(* IEC 61131-3 sources: F100R_S278_Temperville/MyController.device.xml.v3^/Plc Logic.plclogic.xml.v3^/Application.application.xml.v3^/02_Operação, 42 files *)

(* ---- A_EncoderCpu.prg.st ---- *)
PROGRAM A_EncoderCpu

// Encoder Mesa do Forno
IF NOT xRunEncoMForno OR xHomeEncoderForno THEN
	xPresetEncoMForno:=TRUE;
ELSE
	xPresetEncoMforno:=FALSE;
END_IF
dValorEncoderForno:=(-1)*dValorEncoderFornoEntrada;

// Encoder Mesa do Resfriamento
IF NOT xRunEncoMResfr OR xHomeEncoderResfriador THEN
	xPresetEncoMResfr:=TRUE;
ELSE
	xPresetEncoMResfr:=FALSE;
END_IF
dValorEncoderResfriador:=(1)*dValorEncoderResfrEntrada;

// Encoder Dutos Resfriador Superior
IF NOT xRunEncoResfrSup02 OR xHomeEncoderDuctosResfriadorSup02 THEN
	xPresetEncoResfrSup02:=TRUE;
ELSE
	xPresetEncoResfrSup02:=FALSE;
END_IF
dValorEncoderDuctosResfriadorSup02:=(1)*dValorEncoderDuctosResfrSup02Entrada;

// Encoder Dutos Resfriador Inferior
(*IF NOT xRunEncoResfrInf02 OR xHomeEncoderDuctosResfriadorInf02 THEN
	xPresetEncoResfrInf02:=TRUE;
ELSE
	xPresetEncoResfrInf02:=FALSE;
END_IF
dValorEncoderDuctosResfriadorInf02:=(-1)*dValorEncoderDuctosResfrInf02Entrada;
*)
// Encoder Dutos Passagem Superior
(*IF NOT xRunEncoResfrSup01 OR xHomeEncoderDuctosResfriadorSup01 THEN
	xPresetEncoResfrSup01:=TRUE;
ELSE
	xPresetEncoResfrSup01:=FALSE;
END_IF
dValorEncoderDuctosResfriadorSup01:=(1)*dValorEncoderDuctosResfrSup01Entrada;*)

// Encoder Dutos Passagem Inferior
(*IF NOT xRunEncoResfrInf01 OR xHomeEncoderDuctosResfriadorInf01 THEN
	xPresetEncoResfrInf01:=TRUE;
ELSE
	xPresetEncoResfrInf01:=FALSE;
END_IF
dValorEncoderDuctosResfriadorInf01:=(1)*dValorEncoderDuctosResfrInf01Entrada;*)

// Encoder Guilhotina 01
(*IF NOT xRunEncoGuilhotina01 OR xHomeEncoderGuilhotinaResfriador01 THEN
	xPresetEncoGuilhotina01:=TRUE;
ELSE
	xPresetEncoGuilhotina01:=FALSE;
END_IF
dValorEncoderGuilhotinaResfriador01:= (-1)*dValorEncoderGuilhoResfr01Entrada;
*)
// Encoder Guilhotina 01 Superior - Passagem
(*IF NOT xRunEncoGuilhotina01Sup OR xHomeEncoderGuilhotinaResfriador01Sup THEN
	xPresetEncoGuilhotina01Sup:=TRUE;
ELSE
	xPresetEncoGuilhotina01Sup:=FALSE;
END_IF
dValorEncoderGuilhotinaResfriador01Sup:= (1)*dValorEncoderGuilhoResfr01SupEntrada;*)

// Encoder Guilhotina 01 Inferior - Passagem
(*IF NOT xRunEncoGuilhotina01Inf OR xHomeEncoderGuilhotinaResfriador01Inf THEN
	xPresetEncoGuilhotina01Inf:=TRUE;
ELSE
	xPresetEncoGuilhotina01Inf:=FALSE;
END_IF
dValorEncoderGuilhotinaResfriador01Inf:= (1)*dValorEncoderGuilhoResfr01InfEntrada;*)

// Encoder Guilhotina 02
IF NOT xRunEncoGuilhotina02 OR xHomeEncoderGuilhotinaResfriador02 THEN
	xPresetEncoGuilhotina02:=TRUE;
ELSE
	xPresetEncoGuilhotina02:=FALSE;
END_IF
dValorEncoderGuilhotinaResfriador02:= (-1)*dValorEncoderGuilhoResfr02Entrada;

(* ---- A_PrincipalOperacao.prg.st ---- *)
PROGRAM A_PrincipalOperacao
VAR
	HabDesabMotorDuctosInf01: HabilitaDesabilita;
	HabDesabMotorDuctosSup01: HabilitaDesabilita;
	HabDesabMotorDuctosInf02: HabilitaDesabilita;
	HabDesabMotorDuctosSup02: HabilitaDesabilita;
	HabDesabMotorGuilho01: HabilitaDesabilita;
	HabDesabMotorGuilho02: HabilitaDesabilita;

	HabDesabMotorGuilho01Sup: HabilitaDesabilita;
	HabDesabMotorGuilho01Inf: HabilitaDesabilita;
END_VAR

//EncoderMForno();
//EncoderMResfr();
//EncoderResfriInf01();
//EncoderResfriSup01();
//EncoderResfriInf02();
//EncoderResfriSup02();
EncoderModulo01();
EncoderModulo02();
//EncoderModulo03();
//EncoderModulo04();
A_EncoderCpu();
B_Receita();
B_Velocidades();
C_ComandosOperacao();
D_SensoresEntrada();
E_MesaEntrada();
F_BufferForno();
F_MesaForno();
G_BufferResfriamento();
G_BufferTemperaPass();
H_MesaPassagem();
H_MesaResfriador();
H1_Dutos_Oscilantes();
I_MesaSaida();
//J_DuctosResfriadorInf01();
//J_DuctosResfriadorSup01();
//J_DuctosResfriadorInf02();
//J_DuctosResfriadorSup02();
//K_Guilhotina01();
//K_Guilhotina01Sup();
//K_Guilhotina01Inf();
//K_Guilhotina02();
L_EstagiosResfriador();
M_Ventilador01();
//M_Ventilador02();
M_Ventilador03();
//M_Ventilador04();
N_Grades();
//N_MesaBasculante();
O_Portas();
P_ComandosEventos();
//Q_Conveccao();
R_Pressostato();
R_PressostatoAnal();
R_ManometroDifusor();
R_SensorVibracao();
S_ElevacaoForno();
//T_Damper();
T_VenezianaDutPass();
T_VenezianaVentInfPass();
V_VentilacaoPainel();
//X_LimpaResfriador02();

//Habilita/Desabilita Resfriador Inferior 01
(*HabDesabMotorDuctosInf01(Entrada:= xBtDuctosInf01Enable,StatusSaida=> xDuctosInf01Enable);
IF xBtDuctosInf01Enable THEN
	xBtDuctosInf01Enable:=FALSE;
END_IF

IF NOT xDuctosInf01Enable THEN
	J_DuctosResfriadorInf01();
END_IF

xDuctosInf01CheckOk:= xDuctosInf01Enable OR xHomeDuctosResfriadorInf01Ok;
*)

// Habilita/Desabilita Resfriador Superior 01
(*HabDesabMotorDuctosSup01(Entrada:= xBtDuctosSup01Enable,StatusSaida=> xDuctosSup01Enable);
IF xBtDuctosSup01Enable THEN
	xBtDuctosSup01Enable:=FALSE;
END_IF

IF NOT xDuctosSup01Enable THEN
	J_DuctosResfriadorSup01();
END_IF

xDuctosSup01CheckOk:= xDuctosSup01Enable OR xHomeDuctosResfriadorSup01Ok;
*)
// Habilita/Desabilita Resfirador Inferior 02
(*HabDesabMotorDuctosInf02(Entrada:= xBtDuctosInf02Enable,StatusSaida=> xDuctosInf02Enable);
IF xBtDuctosInf02Enable THEN
	xBtDuctosInf02Enable:=FALSE;
END_IF

IF NOT xDuctosInf02Enable THEN
	J_DuctosResfriadorInf02();
END_IF

xDuctosInf02CheckOk:= xDuctosInf02Enable OR xHomeDuctosResfriadorInf02Ok;
*)

// Habilita/Desabilita Resfriador Superior 02
HabDesabMotorDuctosSup02(Entrada:= xBtDuctosSup02Enable,StatusSaida=> xDuctosSup02Enable);
IF xBtDuctosSup02Enable THEN
	xBtDuctosSup02Enable:=FALSE;
END_IF

IF NOT xDuctosSup02Enable THEN
	J_DuctosResfriadorSup02();
END_IF

xDuctosSup02CheckOk:= xDuctosSup02Enable OR xHomeDuctosResfriadorSup02Ok;

// Habilita/Desabilita Guilhotina Resfriador 01
(*HabDesabMotorGuilho01(Entrada:= xBtGuilhotina01Enable,StatusSaida=> xGuilhotina01Enable);
IF xBtGuilhotina01Enable THEN
	xBtGuilhotina01Enable:=FALSE;
END_IF

IF NOT xGuilhotina01Enable THEN
	K_Guilhotina01();
END_IF

xGuilhotina01CheckOk:= xGuilhotina01Enable OR xHomeGuilhotina01Ok;
*)
// Habilita/Desabilita Guilhotina Resfirador 02
HabDesabMotorGuilho02(Entrada:= xBtGuilhotina02Enable,StatusSaida=> xGuilhotina02Enable);
IF xBtGuilhotina02Enable THEN
	xBtGuilhotina02Enable:=FALSE;
END_IF

IF NOT xGuilhotina02Enable THEN
	K_Guilhotina02();
END_IF

xGuilhotina02CheckOk:= xGuilhotina02Enable OR xHomeGuilhotina02Ok;

// Habilita/Desabilita Guilhotina Superior Resfirador 01
(*HabDesabMotorGuilho01Sup(Entrada:= xBtGuilhotina01SupEnable,StatusSaida=> xGuilhotina01SupEnable);
IF xBtGuilhotina01SupEnable THEN
	xBtGuilhotina01SupEnable:=FALSE;
END_IF

IF NOT xGuilhotina01SupEnable THEN
	K_Guilhotina01Sup();
END_IF

xGuilhotina01SupCheckOk:= xGuilhotina01SupEnable OR xHomeGuilhotina01SupOk;*)

// Habilita/Desabilita Guilhotina Inferior Resfirador 01
(*HabDesabMotorGuilho01Inf(Entrada:= xBtGuilhotina01InfEnable,StatusSaida=> xGuilhotina01InfEnable);
IF xBtGuilhotina01InfEnable THEN
	xBtGuilhotina01InfEnable:=FALSE;
END_IF

IF NOT xGuilhotina01InfEnable THEN
	K_Guilhotina01Inf();
END_IF

xGuilhotina01InfCheckOk:= xGuilhotina01InfEnable OR xHomeGuilhotina01InfOk;*)

(* ---- B_Receita.prg.st ---- *)
PROGRAM B_Receita
VAR
	TempoEnvioReceita: TON;
	TempoEnvioReceitaIn: BOOL;
	TempoEnvioReceitaQ: BOOL;
	Index: UINT;
	IndexSoma1: UINT;
	IndexSoma2: UINT;
	IndexSoma3: UINT;
	iSomaRecTemperaturaInferior: INT;
	iSomaRecTemperaturaSuperior: INT;
	iSomaRecPorcentagemInferior: INT;
	iSomaRecPorcentagemSuperior: INT;
	iSomaRecVelocidade01Ventilador01: INT;
	iSomaRecVelocidade02Ventilador01: INT;
	iSomaRecVelocidade01Ventilador02: INT;
	iSomaRecVelocidade02Ventilador02: INT;
	iSomaRecVelocidade01Ventilador03: INT;
	iSomaRecVelocidade02Ventilador03: INT;
	iSomaRecVelocidade01Ventilador04: INT;
	iSomaRecVelocidade02Ventilador04: INT;
	dSomaReceitaSuper: DINT;
END_VAR

IF iHabilitaEscritaReceita=1 THEN
	xReceitaCarregadaOk:=FALSE;
	iEscreverReceita:=1;
	TempoEnvioReceitaIn:=TRUE;
	xBloqueioCargaEnvioRec:=TRUE;
	iHabilitaEscritaReceita:=0;

END_IF

IF iEscreverReceita=1 THEN
	IF 	sEntradaNomedaReceita=sRecNomedaReceita THEN
			xEntradaReenvioRec:=TRUE;
	ELSE
			xEntradaReenvioRec:=FALSE;
	END_IF

	iEntradaEspessuraVidro:=iRecEspessuraVidro;
	rBufferEmissividade:=rRecEmissividade;
	// Parametros de Aquecimento

	rBufferSetTemperaturaInferiorGeral:=rRecTemperaturaInferiorGeral;
	rBufferSetTemperaturaSuperiorGeral:=rRecTemperaturaSuperiorGeral;
	rBufferSetPorcentagemInferiorGeral:=rRecPorcentagemInferiorGeral;
	rBufferSetPorcentagemSuperiorGeral:=rRecPorcentagemSuperiorGeral;

	FOR Index:=1 TO iNumResistencias DO
		rBufferSetTemperaturaSuperior[Index]:=rRecTemperaturaSuperior[Index];
		rBufferSetTemperaturaInferior[Index]:=rRecTemperaturaInferior[Index];
		rBufferSetPorcentagemSuperior[Index]:=rRecPorcentagemSuperior[Index];
		rBufferSetPorcentagemInferior[Index]:=rRecPorcentagemInferior[Index];
	END_FOR

	iBufferTempoPausaResistInf:=iRecTempoPausaResistInf;
	iBufferTempoPausaResistSup:=iRecTempoPausaResistSup;
	iBufferTempoPausa02ResistSup:=iRecTempoPausa02ResistSup;
	iBufferTempoInicioPausa02ResistSup:=iRecTempoInicioPausa02ResistSup;

	iBufferTempoConveccao:=iRecTempoConveccao;

	// Parametros da Mesa do Forno
	iBufferTempoDelayCarga:=iRecTempoDelayCarga;
	iBufferTempoPausaRoletes:=iRecTempoPausaRoletes;
	iBufferTempoAquecimForno:=iRecTempoAquecimForno;
	iBufferTempoPosicaoForno:=iRecTempoPosicaoForno;//////////
	iBufferTempoVelocidadeForno:=iRecTempoVelocidadeForno;////
	iBufferVelocidade01Vaivem:=iRecVelocidade01Vaivem;////////
	iBufferVelocidade02Vaivem:=iRecVelocidade02Vaivem;////////
	iBufferVelocidade03Vaivem:=iRecVelocidade03Vaivem;////////
	iBufferVelocidadeCargaMesadoForno:=iRecVelocidadeCargaMesaForno;////////
	iBufferVelocidadeDescargaMesadoForno:=iRecVelocidadeDescargaMesaForno;/////////
	iBufferCorretorCargaMesaEntrada:=iRecCorretorCargaMesaEntrada;////////

	// Parametros da Mesa do Resfriador

	iBufferTempoResfriamento:=iRecTempoResfriamento;
	iBufferTempoTrocaEstagioResfriamento:=iRecTempoTrocaEstagioResfriamento;
	iBufferTempoTrocaEstagio02Resfriamento:=iRecTempoTrocaEstagio02Resfriamento;

	iBufferVelocidade01Ventilador01:=iRecVelocidade01Ventilador01;
	iBufferVelocidade02Ventilador01:=iRecVelocidade02Ventilador01;
	iBufferVelocidade03Ventilador01:=iRecVelocidade03Ventilador01;

	iBufferVelocidade01Ventilador02:=iRecVelocidade01Ventilador02;
	iBufferVelocidade02Ventilador02:=iRecVelocidade02Ventilador02;
	iBufferVelocidade03Ventilador02:=iRecVelocidade03Ventilador02;

	iBufferVelocidade01Ventilador03:=iRecVelocidade01Ventilador03;
	iBufferVelocidade02Ventilador03:=iRecVelocidade02Ventilador03;
	iBufferVelocidade03Ventilador03:=iRecVelocidade03Ventilador03;

	iBufferVelocidade01Ventilador04:=iRecVelocidade01Ventilador04;
	iBufferVelocidade02Ventilador04:=iRecVelocidade02Ventilador04;
	iBufferVelocidade03Ventilador04:=iRecVelocidade03Ventilador04;

	// Parametros Resfriador 01 Inferior
	iBufferValAltura01ResfriadorInf01:=iRecAltura01ResfriadorInf01;
	iBufferValAltura02ResfriadorInf01:=iRecAltura02ResfriadorInf01;
	iBufferValAltura03ResfriadorInf01:=iRecAltura03ResfriadorInf01;

	// Parametros Resfriador 01 Superior
	iBufferValAltura01ResfriadorSup01:=iRecAltura01ResfriadorSup01;
	iBufferValAltura02ResfriadorSup01:=iRecAltura02ResfriadorSup01;
	iBufferValAltura03ResfriadorSup01:=iRecAltura03ResfriadorSup01;
	iBufferVeneziana:=iRecVeneziana;
	iBufferPassagem:=iRecPassagem;

	// Parametros Resfriador 02 Inferior
	iBufferValAltura01ResfriadorInf02:=iRecAltura01ResfriadorInf02;
	iBufferValAltura02ResfriadorInf02:=iRecAltura02ResfriadorInf02;
	iBufferValAltura03ResfriadorInf02:=iRecAltura03ResfriadorInf02;

	// Parametros Resfriador 02 Superior
	iBufferValAltura01ResfriadorSup02:=iRecAltura01ResfriadorSup02;
	iBufferValAltura02ResfriadorSup02:=iRecAltura02ResfriadorSup02;
	iBufferValAltura03ResfriadorSup02:=iRecAltura03ResfriadorSup02;

	// Parametros Guilhotina 01
	iBufferAlturaGhilhotina01:=iRecAlturaGhilhotina01;

	iBufferAlturaGhilhotina01Sup:=iRecAlturaGhilhotina01Sup;
	iBufferAlturaGhilhotina01Inf:=iRecAlturaGhilhotina01Inf;

	// Parametros Guilhotina 02
	iBufferAlturaGhilhotina02:=iRecAlturaGhilhotina02;

	iBufferCorretorCargaMesaResfriador:=iRecCorretorCargaMesaResfriador;//////////////
	iBufferVelocidadeVaiVemResfriador:=iRecVelocidadeVaiVemResfriador;////////////////////
	iBufferVelocidadeDescargaMesadoResfriador:=iRecVelocidadeDescargaMesaResfriador;////////
	iBufferCorretorCargaMesaSaida:=iRecCorretorCargaMesaSaida;////////////////////

	iRecAjustaAlturaDuctosInf01:=iRecAjustaAlturaDuctosInf01;
	iRecAjustaAlturaDuctosSup01:=iRecAjustaAlturaDuctosSup01;
	iRecAjustaAlturaDuctosInf02:=iRecAjustaAlturaDuctosInf02;
	iRecAjustaAlturaDuctosSup02:=iRecAjustaAlturaDuctosSup02;
	iRecAjustaAlturaGuilho01:=iRecAjustaAlturaGuilho01;
	iRecAjustaAlturaGuilho02:=iRecAjustaAlturaGuilho02;

// Conferencia da Receita
	iSomaRecTemperaturaInferior:=0;
	FOR IndexSoma1:=1	TO iNumResistencias DO
		iSomaRecTemperaturaInferior:=iSomaRecTemperaturaInferior + REAL_TO_INT (rRecTemperaturaInferior[IndexSoma1]);
	END_FOR
	iSomaRecPorcentagemInferior:=0;
	FOR IndexSoma2:=1	TO iNumResistencias DO
		iSomaRecPorcentagemInferior:=iSomaRecPorcentagemInferior + REAL_TO_INT (rRecPorcentagemInferior[IndexSoma2]);
	END_FOR
	iSomaRecTemperaturaSuperior:=0;
	iSomaRecPorcentagemSuperior:=0;
	FOR IndexSoma3:=1	TO iNumResistencias DO
		iSomaRecTemperaturaSuperior:=iSomaRecTemperaturaSuperior + REAL_TO_INT (rRecTemperaturaSuperior[IndexSoma3]);
		iSomaRecPorcentagemSuperior:=iSomaRecPorcentagemSuperior + REAL_TO_INT (rRecPorcentagemSuperior[IndexSoma3]);
	END_FOR

iSomaRecVelocidade01Ventilador01:=iRecVelocidade01Ventilador01/10;
iSomaRecVelocidade02Ventilador01:=iRecVelocidade02Ventilador01/10;
iSomaRecVelocidade01Ventilador02:=iRecVelocidade01Ventilador02/10;
iSomaRecVelocidade02Ventilador02:=iRecVelocidade02Ventilador02/10;
iSomaRecVelocidade01Ventilador03:=iRecVelocidade01Ventilador03/10;
iSomaRecVelocidade02Ventilador03:=iRecVelocidade02Ventilador03/10;
iSomaRecVelocidade01Ventilador04:=iRecVelocidade01Ventilador04/10;
iSomaRecVelocidade02Ventilador04:=iRecVelocidade02Ventilador04/10;

(*
dSomaReceitaClp:=INT_TO_DINT(iRecEspessuraVidro+ REAL_TO_INT (rRecTemperaturaInferiorGeral+rRecTemperaturaSuperiorGeral+
rRecPorcentagemInferiorGeral+rRecPorcentagemSuperiorGeral)+iRecTempoPausaResistInf+iRecTempoPausaResistSup+
iRecTempoConveccao+iRecTempoPausaRoletes+iRecTempoAquecimForno+iRecTempoResfriamento+(iSomaRecVelocidade01Ventilador01)+
(iSomaRecVelocidade02Ventilador01)+(iSomaRecVelocidade01Ventilador02)+(iSomaRecVelocidade02Ventilador02)+
iRecTempoTrocaEstagioResfriamento+iRecAltura01Resfriador+iRecAltura02Resfriador+iRecAlturaGhilhotina+
iSomaRecTemperaturaInferior+iSomaRecTemperaturaSuperior+iSomaRecPorcentagemInferior+iSomaRecPorcentagemSuperior);
*)
	dSomaReceitaSuper:=dSomaReceitaSuperClp;

	sEntradaNomedaReceita:=sRecNomedaReceita;
	xFornoReenvioRec:=xEntradaReenvioRec;
	iReceitaEscritaOk:=1;
	iEscreverReceita:=0;
	xEntradaReenvioRec:=0;
	xReceitaCarregadaOk:=TRUE;
	xBloqueioCargaEnvioRec:=FALSE;
	xReceitaEnviadaEventos:=TRUE;
END_IF
(*
TempoEnvioReceita(IN:=TempoEnvioReceitaIn , PT:=T#15S , Q=>TempoEnvioReceitaQ , ET=> );

IF TempoEnvioReceitaQ THEN
	IF dSomaReceitaClp=dSomaReceitaSuper THEN
		iReceitaEscritaOk:=1;
		iEscreverReceita:=0;
		xReceitaCarregadaOk:=TRUE;
		TempoEnvioReceitaIn:=FALSE;
	ELSE
		iReceitaEscritaFalha:=1;
		iEscreverReceita:=0;
		xReceitaCarregadaOk:=FALSE;
		TempoEnvioReceitaIn:=FALSE;
	END_IF
END_IF
*)

IF (iResfriamentoEspessuraVidro=4 OR iResfriamentoEspessuraVidro=5) THEN
	xEspessuraVidroFino:=TRUE;
	xEspessuraVidroGrosso:=FALSE;
	xBufferValvulaDamperDifusor:=TRUE;
ELSE
	xEspessuraVidroFino:=FALSE;
	xEspessuraVidroGrosso:=TRUE;
	xBufferValvulaDamperDifusor:=FALSE;
END_IF

(* ---- B_Velocidades.prg.st ---- *)
PROGRAM B_Velocidades
VAR
	EntradaForno: EquacaoDaReta;
	FornoPassagem: EquacaoDaReta;
	PassagemResfriamento : EquacaoDaReta;
	ResfriamentoSaida: EquacaoDaReta;
	rVelocidadeMesaEntrada: REAL;
	rVelocidadeCargaMesaForno: REAL;
	rVelocidDescargaMesaForno: REAL;
	rVelocidCargaMesaPassagem: REAL;
	rVelocidDescargaMesaPassagem:REAL;
	rVelocidCargaMesaResfriam: REAL;
	rVelocidDescargaMesaResfr: REAL;
	rVelocidadeMesaSaida: REAL;
	iVelocCargaMesaEntrada: INT;
	iVelocCargaMesaPassagem : INT;
	iVelocCargaResfriador: INT;
	iVelocCargaMesaSaida: INT;
END_VAR

rVelocidadeCargaMesaForno:=INT_TO_REAL(iVelocidadeCargaMesadoForno/1);
rVelocidDescargaMesaForno:=INT_TO_REAL(iVelocidadeDescargaMesadoForno/1);
rVelocidDescargaMesaResfr:=INT_TO_REAL(iVelocidadeDescargaMesadoResfriador/1);

iVelocidadeCargaMesaForno:=REAL_TO_INT(iVelocidadeCargaMesadoForno/10);
iVelocidadeDescargaMesaForno:=REAL_TO_INT(iVelocidadeDescargaMesadoForno/10);
iVelocidadeDescargaMesaResfriador:=REAL_TO_INT(iVelocidadeDescargaMesadoResfriador/10);

EntradaForno(
	rValorY:= rVelocidadeCargaMesaForno/100,
	rPy1:= 25, //Velocidade y1 Inversor Forno
	rPy2:= 45, //Velocidade y2 Inversor Forno
	rPx1:= rVelMesaEntrada25/10, //Velocidade x1 Inversor Entrada
	rPx2:= rVelMesaEntrada45/10, //Velocidade x2 Inversor Entrada
	rValorX=> rVelocidadeMesaEntrada);//Velocidade da Mesa de Entrada

iVelocCargaMesaEntrada:=REAL_TO_INT(rVelocidadeMesaEntrada*10);
iVelocidadeCargaMesaEntrada:=iVelocCargaMesaEntrada+iCorretorCargaMesaEntrada;

FornoPassagem(
	rValorY:= rVelocidDescargaMesaForno/100,
	rPy1:= 25,  //Velocidade y1 Inversor Forno
	rPy2:= 45,  //Velocidade y2 Inversor Forno
	rPx1:= rVelMesaPassagem25/10, //Velocidade x1 Inversor Passagem
	rPx2:= rVelMesaPassagem45/10, //Velocidade x2 Inversor Passagem
	rValorX=> rVelocidCargaMesaPassagem);//Velocidade da Mesa do Resfriamento

iVelocCargaMesaPassagem:=REAL_TO_INT(rVelocidCargaMesaPassagem*10);
iVelocidadeCargaMesaPass:=iVelocCargaMesaPassagem+iCorretorCargaMesaPassagem;

PassagemResfriamento(
	rValorY:= rVelocidDescargaMesaForno/100,
	rPy1:= 25,  //Velocidade y1 Inversor passagem
	rPy2:= 45,  //Velocidade y2 Inversor passagem
	rPx1:= rVelMesaResfriamento25/10, //Velocidade x1 Inversor Resfriador
	rPx2:= rVelMesaResfriamento45/10, //Velocidade x2 Inversor Resfriador
	rValorX=> rVelocidCargaMesaResfriam);//Velocidade da Mesa do Resfriamento

iVelocCargaResfriador:=REAL_TO_INT(rVelocidCargaMesaResfriam*10);
iVelocidadeCargaMesaResfriador:=iVelocCargaResfriador+iCorretorCargaMesaResfriador;

ResfriamentoSaida(
	rValorY:= rVelocidDescargaMesaResfr/10,
	rPy1:= rVelMesaResfriamento25, // Velociade y1 Inversor Resfriador
	rPy2:= rVelMesaResfriamento45, // Velociade y2 Inversor Resfriador
	rPx1:= rVelMesaSaida25, // Velociade x1 Inversor Saída
	rPx2:= rVelMesaSaida45, // Velociade x2 Inversor Saída
	rValorX=> rVelocidadeMesaSaida); // Velocidade da Mesa de Saida

iVelocCargaMesaSaida:=REAL_TO_INT(rVelocidadeMesaSaida);
iVelociadeCargaMesadeSaida:=iVelocCargaMesaSaida+iCorretorCargaMesaSaida;

(* ---- C_ComandosOperacao.prg.st ---- *)
PROGRAM C_ComandosOperacao
VAR
	PassoCmdForno: INT;
	PulsoLedFinalizando: TimerGeneration;
	PulsoLedRestart: TimerGeneration;
	PulsoLedEmEspera: TimerGeneration;
	TonxPausaEmergenciaDelay: TOF;
	TpRestart: TP;
	PulsoPoBtReinicia: PulsoPositivo;
	xLedFornoFinalizando: BOOL;
	xBtRestart: BOOL;
	xPoBtReinicia: BOOL;
	PulsoOperManual: TP;
	PulsoOperAutoma: TP;
	TonOperManual: TON;
	TonOperAutoma: TON;
	TofOperManual: TON;
	TofOperAutoma: TON;

	PulsoPoStartCiclo: PulsoPositivo;
	xFornoEmCicloPulso:	BOOL ;

END_VAR

// SEQUENCIA DE CONTROLE DE OPERAÇÃO

// Seleção Operação ou Stand By

//IF xChStandByOperacao THEN
	xOperacaoHabilitada:=TRUE;
//	xOperacaoStandBy:=FALSE;
(*ELSE
	xOperacaoHabilitada:=FALSE;
	xOperacaoStandBy:=TRUE;
END_IF*)

//Seleção do Modo de Operação Manual ou Automatico
IF xChAutomaticoManual THEN
	xOperacaoManual:=TRUE;
	xOperacaoAutoma:=FALSE;
ELSE
	xOperacaoManual:=FALSE;
	xOperacaoAutoma:=TRUE;
END_IF

PulsoOperManual(IN:= xOperacaoManual, PT:=T#1S , Q=> xPulsoOperacaoManual, ET=> );
PulsoOperAutoma(IN:= xOperacaoAutoma, PT:=T#1S , Q=> xPulsoOperacaoAutoma, ET=> );
TonOperManual(IN:= xOperacaoManual, PT:=T#1S , Q=> xTonOperacaoManual, ET=> );
TonOperAutoma(IN:= xOperacaoAutoma, PT:=T#1S , Q=> xTonOperacaoAutoma, ET=> );
TofOperManual(IN:= xOperacaoManual, PT:=T#1S , Q=> xTofOperacaoManual, ET=> );
TofOperAutoma(IN:= xOperacaoAutoma, PT:=T#1S , Q=> xTofOperacaoAutoma, ET=> );

//Botão de Emergência
xEmergencia:=xBtEmergencia;
// Emergencia para o Supervisório
xBtEmergenciaAcionado:= xBtEmergencia;

IF xEmergencia OR xAlarmeMotorForno THEN
	xPause:=TRUE;
	xRestart:=FALSE;
	xPausaEmergencia:=TRUE;
END_IF
IF NOT xEmergencia THEN
	xPause:=FALSE;
END_IF
(* Reinicio sem Botao Reinicia somente no Reset Alarme *)
IF NOT xEmergencia AND bResetAlmGeral THEN
	xRestart:=TRUE;
	xPausaEmergencia:=FALSE;
ELSE
	xRestart:=FALSE;
END_IF

(* Reinicio com Botão Reinicia Apos Reconhecimento do alarme *)
(*PulsoPoBtReinicia(Entrada:=xBtReinicia, SaidaPulsoPo=>xPoBtReinicia );

IF BtRestart OR xPoBtReinicia THEN
	xBtRestart:=TRUE;
	BtRestart:=FALSE;
ELSE
	xBtRestart:=FALSE;
END_IF

TpRestart(IN:=xBtRestart , PT:=T#500MS , Q=>xBtRestart , ET=> );

IF NOT xEmergencia AND xReleSeguranca AND xBtRestart THEN
	xRestart:=TRUE;
	xPausaEmergencia:=FALSE;
ELSE
	xRestart:=FALSE;
END_IF*)

(*--------- LED RESTART ----------*)

(*PulsoLedRestart.ENABLE:=(xLedStart OR xPausaEmergencia) AND NOT xOperacaoManual;

PulsoLedRestart(ENABLE:= , TIMELOW:=T#500MS , TIMEHIGH:=T#500MS , OUT=>xLedRestart );

(* ----- Informação para Botão Restart do Supervisório -----*)

IF NOT xEmergencia AND xReleSeguranca AND xPausaEmergencia THEN
	xbRestart:=TRUE;
ELSE
	xbRestart:=FALSE;
END_IF*)

TonxPausaEmergenciaDelay(IN:=NOT xReleSeguranca(*xPausaEmergencia*), PT:=T#5000MS , Q=>xPausaEmergenciaTof , ET=> );

(*--------------------------------*)

//Sequencia Ciclo Forno
CASE PassoCmdForno OF

		0:	IF xCmdIniciaCiclo THEN
				PassoCmdForno:=10;
			END_IF

		5:	//xCmdIniciaCiclo:=FALSE;
			PassoCmdForno:=7;

		7: IF xEnergiaOk THEN
				PassoCmdForno:=10;
			ELSE
				PassoCmdForno:=0;
			END_IF

		10: IF xTesteNobreakOk OR xNobreakDesabilitado THEN
				PassoCmdForno:=12;
			END_IF

		12:	uStatusInicioCiclo:=1; // Aguardando Ajustar Dutos
			IF xHomeDuctosResfriadorSup02Ok OR xDuctosSup02Enable THEN
				PassoCmdForno:=15;
			//ELSE
				//PassoCmdForno:=0;
			END_IF

		13:	IF xHomeDuctosResfriadorSup01Ok OR xDuctosSup01Enable THEN
				PassoCmdForno:=15;
			//ELSE
				//PassoCmdForno:=0;
			END_IF

		15:	uStatusInicioCiclo:=2; // Aguardando Ajustar Guilhotina
			IF xHomeGuilhotina02Ok OR xGuilhotina02Enable THEN
				PassoCmdForno:=20;
			//ELSE
				//PassoCmdForno:=0;
			END_IF

		16:	IF xHomeGuilhotina01SupOk OR xGuilhotina01SupEnable THEN
				PassoCmdForno:=17;
			//ELSE
				//PassoCmdForno:=0;
			END_IF

		17:	IF xHomeGuilhotina01InfOk OR xGuilhotina01InfEnable THEN
				PassoCmdForno:=20;
			//ELSE
				//PassoCmdForno:=0;
			END_IF

		20:	uStatusInicioCiclo:=3; // Aguardando Carregar Receita
			IF xReceitaCarregadaOk THEN
				PassoCmdForno:=21;
			//ELSE
				//PassoCmdForno:=0;
			END_IF

		21:	uStatusInicioCiclo:=4; // Aguardando Ligar Resistencias
			IF xLigaResistenciaInferior AND xLigaResistenciaSuperior THEN
				PassoCmdForno:=23;
			//ELSE
				//PassoCmdForno:=0;
			END_IF

		(*22:	uStatusInicioCiclo:=5; // Aguardando Ligar Resistencias Superiores
			IF xLigaResistenciaSuperior THEN
				PassoCmdForno:=23;
			//ELSE
				//PassoCmdForno:=0;
			END_IF*)

		23: uStatusInicioCiclo:=6; // Aguardando Finalizar Aquecimento
			IF uStatusAquecimento=2 THEN // Aquecimento finalizado
				PassoCmdForno:=24;
			//ELSE
				//PassoCmdForno:=0;
			END_IF
			IF xCmFinalizaCiclo OR xSemEnergia THEN(*OR xBtHmiFinalizaCiclo OR xBloqueioAtivo*)
				PassoCmdForno:=40;
			END_IF

		24: xCmdIniciaCiclo:=FALSE;
			xSetTempStandyByInicio:=TRUE;
			PassoCmdForno:=30;

		30:	xFornoEmCiclo:=TRUE;
			IF xCmFinalizaCiclo OR xSemEnergia THEN(*OR xBtHmiFinalizaCiclo OR xBloqueioAtivo*)
				PassoCmdForno:=40;
			END_IF
			IF xAbortaCicloForno THEN
				PassoCmdForno:=200;
			END_IF

		40:	xFornoFinalizando:=TRUE;
			xCmFinalizaCiclo:=FALSE;
			//xBtHmiFinalizaCiclo:=FALSE;
			IF xFornoVazio THEN
				PassoCmdForno:=50;
			END_IF
			IF xAbortaCicloForno THEN
				PassoCmdForno:=200;
			END_IF

		50:	xFornoEmCiclo:=FALSE;
			xFornoFinalizando:=FALSE;
			//xReceitaCarregadaOk:=FALSE;
			xDesligaFimVentilador01:=TRUE;
			xDesligaFimVentilador02:=TRUE;
			xDesligaFimVentilador03:=TRUE;
			xDesligaFimVentilador04:=TRUE;
			PassoCmdForno:=0;

		200:xAbortaCicloForno:=FALSE;
			xFornoFinalizando:=FALSE;
			xBtHmiFinalizaCiclo:=FALSE;
			xFornoEmCiclo:=FALSE;
			xFornoFinalizando:=FALSE;

END_CASE

IF (*NOT xBtFinalizaCiclo OR xBtHmiFinalizaCiclo*)xCmFinalizaCiclo  AND xFornoEmEspera THEN
	//xReceitaCarregadaOk:=FALSE;
	dSomaReceitaClp:=0;
	xReceitaAqiecimCarregadaOk:=FALSE;
	xDesligaFimVentilador01:=TRUE;
	xDesligaFimVentilador02:=TRUE;
	xDesligaFimVentilador03:=TRUE;
	xDesligaFimVentilador04:=TRUE;

	//xBtHmiFinalizaCiclo:=FALSE;
END_IF

xFornoEmEspera:= NOT xFornoEmCiclo AND NOT xFornoFinalizando;

PulsoLedEmEspera(ENABLE:= xFornoEmEspera, TIMELOW:=T#1000MS , TIMEHIGH:=T#1000MS , OUT=>xLedMaqEmEspera );

//xLedMaqEmCiclo:=(xFornoEmCiclo AND NOT xFornoFinalizando) OR xLedFornoFinalizando;

//Sequencia Ciclo Máquina

xMaquinaEmCiclo:= xFornoEmCiclo OR xResfriadorEmCiclo;

xMaquinaEmEspera:= NOT xMaquinaEmCiclo;

// Led Indicação Maquina em Ciclo/Stand-By

PulsoLedFinalizando(ENABLE:= xFornoFinalizando, TIMELOW:=T#500MS , TIMEHIGH:=T#500MS , OUT=>xLedFornoFinalizando );

xLedMaqEmCiclo:=(xFornoEmCiclo AND NOT xFornoFinalizando) OR xLedFornoFinalizando OR xLedMaqEmEspera;

// Libera Ajuste da Altura dos Ductos e da Guilhotina

IF iRecAjustaAlturaDuctosInf01=1 AND xFornoEmCiclo AND xReceitaCarregadaOk THEN
	xBtRecAjustaAlturaDuctosInf01:=TRUE;
	iRecAjustaAlturaDuctosInf01:=0;
END_IF

IF iRecAjustaAlturaDuctosSup01=1 AND xFornoEmCiclo AND xReceitaCarregadaOk THEN
	xBtRecAjustaAlturaDuctosSup01:=TRUE;
	iRecAjustaAlturaDuctosSup01:=0;
END_IF

IF iRecAjustaAlturaDuctosInf02=1 AND xFornoEmCiclo AND xReceitaCarregadaOk THEN
	xBtRecAjustaAlturaDuctosInf02:=TRUE;
	iRecAjustaAlturaDuctosInf02:=0;
END_IF

IF iRecAjustaAlturaDuctosSup02=1 AND xFornoEmCiclo AND xReceitaCarregadaOk THEN
	xBtRecAjustaAlturaDuctosSup02:=TRUE;
	iRecAjustaAlturaDuctosSup02:=0;
END_IF

IF iRecAjustaAlturaGuilho01=1 AND xFornoEmCiclo AND xReceitaCarregadaOk THEN
	xBtRecAjustaGuilhotina01:=TRUE;
	iRecAjustaAlturaGuilho01:=0;
END_IF

IF iRecAjustaAlturaGuilho02=1 AND xFornoEmCiclo AND xReceitaCarregadaOk THEN
	xBtRecAjustaGuilhotina02:=TRUE;
	iRecAjustaAlturaGuilho02:=0;
END_IF

// Auto Home Motores Dutos e Guilhotina
PulsoPoStartCiclo(Entrada:= xFornoEmCiclo, SaidaPulsoPo=> xFornoEmCicloPulso);

IF xFornoEmCicloPulso AND NOT xFornoEmCiclocomCarga AND NOT xResfriadorEmCiclo THEN
	xAutoHomeResfInf02	:= TRUE ;
	xAutoHomeResfSup02	:= TRUE ;
	xAutoHomeGuilho01	:= TRUE ;
	xAutoHomeGuilho02	:= TRUE ;
END_IF

IF xOperacaoManual THEN
	PassoCmdForno:=0;
	xAbortaCicloForno:=FALSE;
	xFornoFinalizando:=FALSE;
	xBtHmiFinalizaCiclo:=FALSE;
	xFornoEmCiclo:=FALSE;
	xFornoFinalizando:=FALSE;
	//xReceitaCarregadaOk:=FALSE;
	dSomaReceitaClp:=0;
	iRecAjustaAlturaDuctosInf01:=0;
	iRecAjustaAlturaDuctosSup01:=0;
	iRecAjustaAlturaDuctosInf02:=0;
	iRecAjustaAlturaDuctosSup02:=0;
	iRecAjustaAlturaGuilho01:=0;
	iRecAjustaAlturaGuilho02:=0;
	xBtRecAjustaAlturaDuctosSup01:=FALSE;
	xBtRecAjustaAlturaDuctosInf01:=FALSE;
	xBtRecAjustaAlturaDuctosSup02:=FALSE;
	xBtRecAjustaAlturaDuctosInf02:=FALSE;
	xBtRecAjustaGuilhotina01:=FALSE;
	xBtRecAjustaGuilhotina02:=FALSE;

	xPausaEmergencia:=FALSE;
	xAutoHomeResfInf02	:= FALSE ;
	xAutoHomeResfSup02	:= FALSE ;
	xAutoHomeGuilho01	:= FALSE ;
	xAutoHomeGuilho02	:= FALSE ;
END_IF

(* ---- E_MesaEntrada.prg.st ---- *)
PROGRAM E_MesaEntrada
VAR
	PassoMesaEntrada: INT;
	PassoPauseEntrada: INT;
	PassoAlmEntrada: INT;
	PassoManualEntrada: INT;
	///Blocos Nativos
	PulsaLedCarga: TimerGeneration;
	PulsoRetornaSensor: TOF;
	TempoLimRetornoSensor: TON;
	TonDelayMovEntrada: TON;
	TempoDelayCarga: Temporizador;
	TempoAposSairSensor: TON;
	TempoAposSairSensorIn: BOOL;
	TempoAposSairSensorQ: BOOL;
	TonAbortaCargaVazio: TON;
	TonAbortaCargaVazioIn: BOOL;
	TonAbortaCargaVazioQ: BOOL;
	PulsaLedCargaIn: BOOL;
	PulsaLedCargaQ: BOOL;
	///Blocos Criados
	PulsoPoChAvanco: PulsoPositivo;
	PulsoNeChAvanco: PulsoNegativo;
	xChAvancaMesaEntradaPo: BOOL;
	xChAvancaMesaEntradaNe: BOOL;
	xAvancoMesaEntrada: BOOL;
	xRecuoMesaEntrada: BOOL;
	xAvancoJogMesaEntrada: BOOL;
	xRecuoJogMesaEntrada: BOOL;
	xCmdAvancoMesaEntrada: BOOL;
	xCarregaFornoManual: BOOL;
	xCarregaFornoAuto: BOOL;
	///xCarregamentoHabilitado: BOOL;
	xLigaCargaForno: BOOL;
	xCarregandoMesaEntrada: BOOL;
	xSeguraCarga: BOOL;
	xCarregaForno: BOOL;
	xRetornoSensor: BOOL;
	xFornoProntoReceber: BOOL;
	iVelocidadeMesaEntrada: INT;
	///xCargaFornoEmAutomatico: BOOL;
	xCargaFornoEmManual: BOOL;
	xPulsoRetornaSensor: BOOL;
	xDelayMovEntrada: BOOL;
	xFimDelayCarregamento: BOOL;
	xDelayCargaOn: BOOL;
	xTempoDiferencaCargas: BOOL;
	xDesligaCargaVazia: BOOL;
	RPM: INT;
	HZ: INT;
END_VAR

// JOG DA MESA DE ENTRADA
(*Avanço*)
PulsoPoChAvanco(Entrada:= xChAvancaMesaEntrada, SaidaPulsoPo=>xChAvancaMesaEntradaPo );
PulsoNeChAvanco(Entrada:= xChAvancaMesaEntrada, SaidaPulsoNe=>xChAvancaMesaEntradaNe );

xCmdAvancoMesaEntrada:=(xChAvancaMesaEntradaPo OR xCmdAvancoMesaEntrada) AND NOT xChAvancaMesaEntradaNe AND NOT xSensorEntrada;

IF xCmdAvancoMesaEntrada AND NOT xCarregandoForno AND NOT xRetornandoForno AND NOT xSensorEntrada (*AND NOT xPausaEmergencia*) AND xTonOperacaoAutoma THEN
	xAvancoJogMesaEntrada:=TRUE;
ELSE
	xAvancoJogMesaEntrada:=FALSE;
END_IF

PulsoRetornaSensor(IN:=xChAvancaMesaEntradaPo , PT:=T#100MS , Q=>xPulsoRetornaSensor , ET=> );
IF (xPulsoRetornaSensor OR xBtHabilitaCarregamento OR xRecargaForno) AND xSensorEntrada  THEN
	xRetornoSensor:=TRUE;
(*ELSE
	xRetornoSensor:=FALSE;*)
END_IF
// Tempo Limite de retorno pelo sensor
TempoLimRetornoSensor(IN:=xRetornoSensor, PT:=T#6S , Q=> , ET=> );

TempoAposSairSensorIn:=NOT xSensorEntrada;
TempoAposSairSensor(IN:=TempoAposSairSensorIn, PT:=T#3S , Q=>TempoAposSairSensorQ , ET=> );

IF TempoAposSairSensorQ OR TempoLimRetornoSensor.Q  THEN
	xRetornoSensor:=FALSE;
END_IF

(*Recuo*)
IF (xChRecuaMesaEntrada OR xRetornoSensor) AND NOT xCarregandoForno AND NOT xRetornandoForno (*AND NOT xPausaEmergencia*) THEN
	xRecuoJogMesaEntrada:=TRUE;
ELSE
	xRecuoJogMesaEntrada:=FALSE;
END_IF

//PRE CONDIÇÕES PARA CARREGAMENTO
(*xTempoDiferencaCargas*)
// Tempo de Restante de Resfriamento Maior que Programado de Forno -> Segura Carregamento
IF (iTempoResfriamentoRestante>=iTempoAquecimForno-10 ) THEN
	xTempoDiferencaCargas:=TRUE;
ELSE
	xTempoDiferencaCargas:=FALSE;
END_IF
IF xTempoDiferencaCargas AND xResfriadorEmCiclo(*xResfriadorCheio*) THEN
	xSeguraCarga:= TRUE;
ELSE
	xSeguraCarga:= FALSE;
END_IF;
// Habilita Carregamento Automatico
IF xBtHabilitaCarregamento AND xFornoEmCiclo AND NOT xBloqueioCargaEnvioRec AND NOT xFornoFinalizando AND NOT xAvancoJogMesaEntrada AND NOT xRecuoJogMesaEntrada AND NOT xSensorEntrada (**)AND NOT xAlarmeMotorForno (**)AND NOT xAlarmeMotorEntrada THEN
	xCarregamentoHabilitado:=TRUE;
	xCargaFornoEmAutomatico:=TRUE;

END_IF
// Carregamento Manual
IF xBtHabilitaCarregamento AND xFornoEmCiclo AND NOT xBloqueioCargaEnvioRec AND NOT xFornoFinalizando AND xFornoVazio THEN
	xCarregaFornoManual:=TRUE;

END_IF

IF xRecargaForno AND xCarregamentoHabilitado AND NOT xSensorEntrada THEN
	xCarregaFornoAuto:=TRUE;
	xCargaFornoEmAutomatico:=TRUE;
END_IF
IF xRecargaForno THEN
	xRecargaForno:=FALSE;
END_IF

// Tempo de atraso no Carregamento automatico do forno
TempoDelayCarga(
	IniciaTempo:= xDelayCargaForno,
	AbortaTempo:= xOperacaoManual,
	SetPointTempo:= iTempoDelayCarga,
	FimTempo:= xFimDelayCarregamento,
	TempoDecorrido=> iTempoDelayCargaDecorrido,
	TempoRestante=> );

IF xDelayCargaForno THEN
	xDelayCargaOn:=TRUE;
	xDelayCargaForno:=FALSE;
END_IF

IF xFimDelayCarregamento THEN
	xDelayCargaOn:=FALSE;
END_IF

IF (xCarregaFornoAuto OR xCarregaFornoManual) AND NOT  xSeguraCarga AND NOT xDelayCargaOn AND (sEntradaNomedaReceita=sFornoNomedaReceita) THEN
	xCarregaForno:=TRUE;
	xCarregaFornoAuto:=FALSE;
	xCarregaFornoManual:=FALSE;
END_IF

IF  xCarregaForno AND xCarregamentoHabilitado AND NOT xSeguranca THEN
	xLigaCargaForno:=TRUE;
	xCarregaForno:=FALSE;
	xCarregamentoHabilitado:=FALSE;
	xFimDelayCarregamento:=FALSE;
END_IF
IF xSeguranca THEN
	xLigaCargaForno:=FALSE;
	xCarregaForno:=FALSE;
	xCarregamentoHabilitado:=FALSE;
END_IF

IF NOT xCarregandoForno AND xFornoEmCiclo AND NOT xBloqueioCargaEnvioRec AND NOT xFornoFinalizando (**)AND NOT xAlarmeMotorForno (**)and not xAlarmeMotorEntrada THEN
	xFornoProntoReceber:=TRUE;
ELSE
	xFornoProntoReceber:=FALSE;
END_IF

PulsaLedCarga(ENABLE:= xFornoProntoReceber, TIMELOW:=T#500MS , TIMEHIGH:=T#500MS , OUT=>PulsaLedCargaQ );
xLedCargaForno:=(xCargaFornoEmAutomatico OR PulsaLedCargaQ) AND NOT xCarregandoForno;

xCargaEmAutomatico:=xCargaFornoEmAutomatico;

//Aborta Carregamento Automático
IF (((xAvancoJogMesaEntrada OR xRecuoJogMesaEntrada ) AND NOT  xCarregandoForno AND NOT xRetornandoForno) OR NOT xFornoEmCiclo (*OR xAlarmePortaEntradaForno OR xAlarmeMotorEntrada OR xAlarmeMotorForno*)) AND xIniciaCargaMesaEntrada THEN
	xFornoEmCicloComCarga:=FALSE;//
END_IF
IF ((xAvancoJogMesaEntrada OR xRecuoJogMesaEntrada ) AND NOT  xCarregandoForno AND NOT xRetornandoForno) OR NOT xFornoEmCiclo (*OR xAlarmePortaEntradaForno OR xAlarmeMotorEntrada OR xAlarmeMotorForno*) THEN
	xCarregaFornoAuto:=FALSE;
	xCarregaFornoManual:=FALSE;
	xCarregamentoHabilitado:=FALSE;
	PassoMesaEntrada:=0;
	xCargaFornoEmAutomatico:=FALSE;
    xPortaEntradaForno:=FALSE;
	xIniciaCargaMesaEntrada:=FALSE; //->TASK/MesaForno
	xCarregandoMesaEntrada:=FALSE;
	xLigaCargaForno:=FALSE;//

	xFimCarregamentoMesaEntrada:=FALSE;(**)
	xFimCargaMesaEntrada:=FALSE;(**)
	xRetornaMesaEntrada:=FALSE;(**)

	xRecuoMesaEntrada:=FALSE; (*teste*)
	xFimRetornoMesaEntrada:=FALSE;(*teste*)
	xAvancoMesaEntrada:=FALSE;(*teste*)

END_IF

// SEQUENCIA DE CARREGAMENTO
TonDelayMovEntrada(IN:= xInvMesaEntradaHabilitado, PT:=T#1S , Q=> xDelayMovEntrada, ET=> );

CASE PassoMesaEntrada OF

		0:	IF xLigaCargaForno THEN
				IF xMotorFornoLigado THEN
					PassoMesaEntrada:=1;
				END_IF
				IF xPause THEN
					PassoPauseEntrada:=0;
					PassoMesaEntrada:=200;
				END_IF
				IF xAlarmeMotorEntrada OR xAlarmeMotorForno OR xAlarmeGeralEncoderMeForno THEN
					PassoMesaEntrada:=200;
				END_IF
			END_IF

		1: 	xLigaCargaForno:=FALSE;
			PassoMesaEntrada:=2;

		2:	xFornoEmCicloComCarga:=TRUE;
			PassoMesaEntrada:=3;

		3:	iVelocidadeMesaForno:= iVelocidadeCargaMesaForno;(*Velocidade Carga Forno*)
			PassoMesaEntrada:=4;

		4:	PassoMesaEntrada:=5;

		5:	PassoMesaEntrada:=6;

		6:	IF iVelocidadeCargaMesaForno= iFrequenciaMotorMesaForno THEN
				PassoMesaEntrada:=10;
			ELSE
				PassoMesaEntrada:=2;
			END_IF

		10:	xPortaEntradaForno:=TRUE;
			PassoMesaEntrada:=20;

		20:	IF xSensorPortaEntrada THEN
				PassoMesaEntrada:=30;
			END_IF
			IF xPause THEN
				PassoPauseEntrada:=0;
				PassoMesaEntrada:=200;
			END_IF
			IF xAlarmeMotorEntrada OR xAlarmeMotorForno OR xAlarmeGeralEncoderMeForno OR xAlarmePortaEntradaForno THEN
				PassoMesaEntrada:=200;
			END_IF

		30:	iVelocidadeMesaEntrada:= iVelocidadeCargaMesaEntrada;(*Velocidade Carga Mesa Entrada*)
			PassoMesaEntrada:=31;

		31:	xAvancoMesaEntrada:=TRUE;
			PassoMesaEntrada:=40;

   		40:	IF xCarregandoForno THEN
				PassoMesaEntrada:=50;
			ELSE
				PassoMesaEntrada:=44;
			END_IF

		44:	xIniciaCargaMesaEntrada:=TRUE; //->TASK/MesaForno
			xCarregandoMesaEntrada:=TRUE;
			TonAbortaCargaVazioIn:=TRUE;
			PassoMesaEntrada:=45;

		45:	IF xIniciaCargaForno THEN
				PassoMesaEntrada:=46;
			END_IF
			IF xPause THEN
				PassoPauseEntrada:=0;
				PassoMesaEntrada:=200;
			END_IF
			IF xAlarmeMotorEntrada OR xAlarmeMotorForno OR xAlarmeGeralEncoderMeForno OR xAlarmePortaEntradaForno THEN
				PassoMesaEntrada:=200;
			END_IF
			IF TonAbortaCargaVazioQ  THEN
				PassoMesaEntrada:=200;
			END_IF

		46: TonAbortaCargaVazioIn:=FALSE;
			PassoMesaEntrada:=50;

		50:	IF xFimCarregamentoMesaEntrada THEN //<- TASK/MesaForno //
				PassoMesaEntrada:=55;
			END_IF
			IF xPause THEN
				PassoPauseEntrada:=30;
				PassoMesaEntrada:=300;
			END_IF
			IF xAlarmeMotorEntrada OR xAlarmeMotorForno OR xAlarmeGeralEncoderMeForno OR xAlarmePortaEntradaForno THEN
				PassoAlmEntrada:=30;
				PassoMesaEntrada:=400;
			END_IF

		55:	xAvancoMesaEntrada:=FALSE;
			PassoMesaEntrada:=56;

		56:	xCargaFornoEmAutomatico:=FALSE;
			xLigaCargaForno:=FALSE;
			xFimCarregamentoMesaEntrada:=FALSE;
			xCarregandoMesaEntrada:=FALSE;
			PassoMesaEntrada:=60;

		60: PassoMesaEntrada:=70;

		70:	IF xFimCargaMesaEntrada THEN //<- TASK/MesaForno
				PassoMesaEntrada:=120;
			END_IF;
			IF xRetornaMesaEntrada THEN //<- TASK/MesaForno
				PassoMesaEntrada:=80;
			END_IF

		80:	xLigaCargaForno:=FALSE;
			xRetornaMesaEntrada:=FALSE;
			iVelocidadeMesaEntrada:= 1*iVelocidadeCargaMesaEntrada;(*iVelRetornoMesaEntrada;Velocidade Retorno Mesa Entrada*)
			PassoMesaEntrada:=81;

		81:	xRecuoMesaEntrada:=TRUE;
			PassoMesaEntrada:=90;

		90:	IF xFimRetornoMesaEntrada THEN //<- TASK/MesaForno
				PassoMesaEntrada:=100;
			END_IF
			IF xPause THEN
				PassoPauseEntrada:=80;
				PassoMesaEntrada:=300;
			END_IF
			IF xAlarmeMotorEntrada OR xAlarmeMotorForno OR xAlarmeGeralEncoderMeForno OR xAlarmePortaEntradaForno THEN
				PassoAlmEntrada:=80;
				PassoMesaEntrada:=400;
			END_IF

		100:PassoMesaEntrada:=101;

		101:xRecuoMesaEntrada:=FALSE;
			PassoMesaEntrada:=110;

		110:xFimRetornoMesaEntrada:=FALSE;
		    xPortaEntradaForno:=FALSE;
			PassoMesaEntrada:=0;

		120:xFimCargaMesaEntrada:=FALSE;
		    xPortaEntradaForno:=FALSE;
			PassoMesaEntrada:=0;

		//Alarmes
		200:xRecuoMesaEntrada:=FALSE;
			xAvancoMesaEntrada:=FALSE;
			PassoMesaEntrada:=201;

		201:PassoMesaEntrada:=202;

		202: xLigaCargaForno:=FALSE;
			 xPortaEntradaForno:=FALSE;
			 xFornoEmCicloComCarga:=FALSE;
			 xCargaFornoEmAutomatico:=FALSE;
			 xIniciaCargaMesaEntrada:=FALSE;
			 xCarregandoMesaEntrada:=FALSE;
			 PassoMesaEntrada:=0;

		// Emergência Pausa/Reinicio
		300:xRecuoMesaEntrada:=FALSE;
			xAvancoMesaEntrada:=FALSE;
			PassoMesaEntrada:=301;

		301:PassoMesaEntrada:=302;

		302:IF xRestart THEN
				PassoMesaEntrada:=303;
			END_IF

		303:PassoMesaEntrada:=PassoPauseEntrada;

		// Alarme Motor Parada/Reinicio
		400:xRecuoMesaEntrada:=FALSE;
			xAvancoMesaEntrada:=FALSE;
			PassoMesaEntrada:=401;

		401:PassoMesaEntrada:=402;

		402:IF xRestart AND iCanOpenInverMesaEntraStateOk THEN
				PassoMesaEntrada:=PassoAlmEntrada;
			END_IF

END_CASE

// MOVIMENTAÇÃO PELO COMANDO ENTRADAS DIGITAIS DO INVERSOR
// Comando e Direção
xMotorMesaEntradaAvanco:= xAvancoMesaEntrada OR xAvancoJogMesaEntrada;
xMotorMesaEntradaRecuo:= xRecuoMesaEntrada OR xRecuoJogMesaEntrada;

InversorMesaEntrada.i_xAvanco:=xMotorMesaEntradaAvanco;
InversorMesaEntrada.i_xRecuo:=xMotorMesaEntradaRecuo;

// Velocidade
IF xAvancoJogMesaEntrada OR xRecuoJogMesaEntrada THEN
	IF xRetornoSensor THEN
		InversorMesaEntrada.i_iFreqRef:=50;
	ELSE
		InversorMesaEntrada.i_iFreqRef:=iVelocidadeJogMesaEntrada;
	END_IF
ELSE
	InversorMesaEntrada.i_iFreqRef:=iVelocidadeMesaEntrada;
END_IF
//--------------------------------------------------------------------------\\

IF xOperacaoManual THEN
	PassoMesaEntrada:=0;
	PassoPauseEntrada:=0;
	PassoAlmEntrada:=0;
	xCarregamentoHabilitado:=FALSE;
	xCargaFornoEmAutomatico:=FALSE;
	xCarregaFornoManual:=FALSE;
	xCarregaFornoAuto:=FALSE;
	xCarregaForno:=FALSE;
	xLigaCargaForno:=FALSE;
	xIniciaCargaMesaEntrada:=FALSE;
	xCarregandoMesaEntrada:=FALSE;
	xFimCarregamentoMesaEntrada:=FALSE;
	xFimCargaMesaEntrada:=FALSE;
	xRetornaMesaEntrada:=FALSE;
	xFimRetornoMesaEntrada:=FALSE;
	xDelayCargaForno:=FALSE;
	xFimDelayCarregamento:=FALSE;
	xDelayCargaOn:=FALSE;
	xBloqueioCargaEnvioRec:=FALSE;

	xAvancoJogMesaEntrada:=FALSE;
	xRecuoJogMesaEntrada:=FALSE;
	xAvancoMesaEntrada:=FALSE;
	xRecuoMesaEntrada:=FALSE;

END_IF

TonAbortaCargaVazio(IN:= TonAbortaCargaVazioIn, PT:=T#20S , Q=>  TonAbortaCargaVazioQ, ET=>);
IF TonAbortaCargaVazioQ OR xOperacaoManual THEN
	TonAbortaCargaVazioIn:=FALSE;
END_IF

(* ---- F_BufferForno.prg.st ---- *)
PROGRAM F_BufferForno
VAR
	Index: INT;
	iEscreverReceitaForno: INT;
END_VAR

IF ((sEntradaNomedaReceita<>sFornoNomedaReceita) OR xFornoReenvioRec) AND xFornoVazio THEN
	iEscreverReceitaForno:=1;
END_IF

IF iEscreverReceitaForno=1 THEN
	iFornoEspessuraVidro:=iEntradaEspessuraVidro;
	// Parametros de Aquecimento

	rSetTemperaturaInferiorGeral:=rBufferSetTemperaturaInferiorGeral;
	rSetTemperaturaSuperiorGeral:=rBufferSetTemperaturaSuperiorGeral;
	rSetPorcentagemInferiorGeral:=rBufferSetPorcentagemInferiorGeral;
	rSetPorcentagemSuperiorGeral:=rBufferSetPorcentagemSuperiorGeral;

	rSetTemperaturaInferiorGeralAux:=rBufferSetTemperaturaInferiorGeral;
	rSetTemperaturaSuperiorGeralAux:=rBufferSetTemperaturaSuperiorGeral;
	rSetPorcentagemInferiorGeralAux:=rBufferSetPorcentagemInferiorGeral;
	rSetPorcentagemSuperiorGeralAux:=rBufferSetPorcentagemSuperiorGeral;

	FOR Index:=1	TO iNumResistencias DO
		rSetTemperaturaSuperior[Index]:=rBufferSetTemperaturaSuperior[Index];
		rSetTemperaturaInferior[Index]:=rBufferSetTemperaturaInferior[Index];
		rSetPorcentagemSuperior[Index]:=rBufferSetPorcentagemSuperior[Index];
		rSetPorcentagemInferior[Index]:=rBufferSetPorcentagemInferior[Index];
	END_FOR

	iTempoPausaResistInf:=iBufferTempoPausaResistInf;
	iTempoPausaResistSup:=iBufferTempoPausaResistSup;
	iTempoPausa02ResistSup:=iBufferTempoPausa02ResistSup;
	iTempoInicioPausa02ResistSup:=iBufferTempoInicioPausa02ResistSup;

	iTempoConveccao:=iBufferTempoConveccao;

	// Parametros da Mesa do Forno
	iTempoDelayCarga:=iBufferTempoDelayCarga;
	iTempoPausaRoletes:=iBufferTempoPausaRoletes;
	iTempoAquecimForno:=iBufferTempoAquecimForno;
	iTempoPosicaoForno:=iBufferTempoPosicaoForno;//////////
	iTempoVelocidadeForno:=iBufferTempoVelocidadeForno;////
	iVelocidade01Vaivem:=iBufferVelocidade01Vaivem;////////
	iVelocidade02Vaivem:=iBufferVelocidade02Vaivem;////////
	iVelocidade03Vaivem:=iBufferVelocidade03Vaivem;////////
	iVelocidadeCargaMesadoForno:=iBufferVelocidadeCargaMesadoForno;////////
	iVelocidadeDescargaMesadoForno:=iBufferVelocidadeDescargaMesadoForno;/////////
	iCorretorCargaMesaEntrada:=iBufferCorretorCargaMesaEntrada;////////

	// Parametros da Mesa do Resfriador
	rBuffer02Emissividade:=rBufferEmissividade;

	iBuffer02TempoResfriamento:=iBufferTempoResfriamento;
	iBuffer02TempoTrocaEstagioResfriamento:=iBufferTempoTrocaEstagioResfriamento;
	iBuffer02TempoTrocaEstagio02Resfriamento:=iBufferTempoTrocaEstagio02Resfriamento;

	//iBuffer02Velocidade01Ventilador01:=iBufferVelocidade01Ventilador01;
	iVelocidade01Ventilador01:=iBufferVelocidade01Ventilador01;
	iBuffer02Velocidade02Ventilador01:=iBufferVelocidade02Ventilador01;
	iBuffer02Velocidade03Ventilador01:=iBufferVelocidade03Ventilador01;

	iBuffer02Velocidade01Ventilador02:=iBufferVelocidade01Ventilador02;
	iBuffer02Velocidade02Ventilador02:=iBufferVelocidade02Ventilador02;
	iBuffer02Velocidade03Ventilador02:=iBufferVelocidade03Ventilador02;

	iBuffer02Velocidade01Ventilador03:=iBufferVelocidade01Ventilador03;
	iBuffer02Velocidade02Ventilador03:=iBufferVelocidade02Ventilador03;
	iBuffer02Velocidade03Ventilador03:=iBufferVelocidade03Ventilador03;

	iBuffer02Velocidade01Ventilador04:=iBufferVelocidade01Ventilador04;
	iBuffer02Velocidade02Ventilador04:=iBufferVelocidade02Ventilador04;
	iBuffer02Velocidade03Ventilador04:=iBufferVelocidade03Ventilador04;

	// Parametros Resfriador 01 Inferior
	iBuffer02ValAltura01ResfriadorInf01:=iBufferValAltura01ResfriadorInf01;
	iBuffer02ValAltura02ResfriadorInf01:=iBufferValAltura02ResfriadorInf01;
	iBuffer02ValAltura03ResfriadorInf01:=iBufferValAltura03ResfriadorInf01;

	// Parametros Resfriador 01 Superior
	iBuffer02ValAltura01ResfriadorSup01:=iBufferValAltura01ResfriadorSup01;
	iBuffer02ValAltura02ResfriadorSup01:=iBufferValAltura02ResfriadorSup01;
	iBuffer02ValAltura03ResfriadorSup01:=iBufferValAltura03ResfriadorSup01;
	iBuffer02Veneziana:=iBufferVeneziana;
	iBuffer02Passagem:=iBufferPassagem;

	// Parametros Resfriador 02 Inferior
	iBuffer02ValAltura01ResfriadorInf02:=iBufferValAltura01ResfriadorInf02;
	iBuffer02ValAltura02ResfriadorInf02:=iBufferValAltura02ResfriadorInf02;
	iBuffer02ValAltura03ResfriadorInf02:=iBufferValAltura03ResfriadorInf02;

	// Parametros Resfriador 02 Superior
	iBuffer02ValAltura01ResfriadorSup02:=iBufferValAltura01ResfriadorSup02;
	iBuffer02ValAltura02ResfriadorSup02:=iBufferValAltura02ResfriadorSup02;
	iBuffer02ValAltura03ResfriadorSup02:=iBufferValAltura03ResfriadorSup02;

	// Parametros Guilhotina 01
	iBuffer02AlturaGhilhotina01:=iBufferAlturaGhilhotina01;

	iBuffer02AlturaGhilhotina01Sup:=iBufferAlturaGhilhotina01Sup;
	iBuffer02AlturaGhilhotina01Inf:=iBufferAlturaGhilhotina01Inf;

	// Parametros Guilhotina 02
	iBuffer02AlturaGhilhotina02:=iBufferAlturaGhilhotina02;

	iBuffer02CorretorCargaMesaResfriador:=iBufferCorretorCargaMesaResfriador;
	iBuffer02VelocidadeVaiVemResfriador:=iBufferVelocidadeVaiVemResfriador;
	iBuffer02VelocidadeDescargaMesadoResfriador:=iBufferVelocidadeDescargaMesadoResfriador;
	iBuffer02CorretorCargaMesaSaida:=iBufferCorretorCargaMesaSaida;

	sFornoNomedaReceita:=sEntradaNomedaReceita;
	xResfriamentoReenvioRec:=xFornoReenvioRec;
	iEscreverReceitaForno:=0;
	xFornoReenvioRec:=0;
END_IF

IF iFornoEspessuraVidro = 4 THEN
	xEspessuraVidroFino:=TRUE;
	xEspessuraVidroGrosso:=FALSE;
ELSE
	xEspessuraVidroFino:=FALSE;
	xEspessuraVidroGrosso:=TRUE;
END_IF

(* ---- F_MesaForno.prg.st ---- *)
PROGRAM F_MesaForno
VAR
	///Passo da Execução da Movimentação do Forno
	PassoMesaForno: INT;
	///Passo da Execução da Movimentação do Forno
	PassoIniciaForno: INT;
	PassoAlmIniForno: INT;
	PassoManualForno: INT;
	PassoEmergenciaForno: INT;
	PassoPauseForno: INT;
	PassoAlmMesaForno: INT;
	PassoPauseIniForno: INT;
	PassoVelVaivem: INT;
	////////
	PassoPosVaivem: INT;
	///////
	SetRampasForno: GIATV.SetDriveRamp_ATV;
	TpSairForno: TP;
	TonParadaSemEner: TON;
	TonDelayMovForno: TON;
	TonParadaSemEnerIn: BOOL;
	TonParadaSemEnerQ: BOOL;
	TonParadaSemEnerEt: TIME;
	TonAutoResetMotorForno: TON;
	TonAutoResetMotorFornoIn: BOOL;
	TonAutoResetMotorFornoQ: BOOL;
	TonIniVelStd: TON;
	TonIniVelStdIn: BOOL;
	TonIniVelStdQ: BOOL;
	///Bloco Conta Tempo de Pausa dos Roletes
	TempoPausaRoletes: Temporizador;
	///Bloco Conta Tempo de Permanecia no Forno
	TempoAquecimForno: Temporizador;
	TempoTrocaVelocidade: Temporizador;
	///////////////////////////////////////////
	TempoTrocaPosicao: Temporizador;
	///////////////////////////////////////////
	TamanhoCarga: ComprimentoCarga;
	///Bloco Calcula Posições de Paradas da Carga
	CalculosMesaForno: CalculosForno;
	///Bloco Converte Milimetro em Pulsos
	ConversorMilimPul: MmConversorPulso;
	///Bloco Converte Pulsos em Milimetros
	ConversorPulMilim: PulsoConversorMm;
	///Bloco Seleciona Pulsos para Vidro Fino ou Grosso
	SelecaoPulsos: BlocoSelecaoEspessura;
	xExecutaSetRampasForno: BOOL;
	dAceleracaoMesaForno: DINT;
	dDesaceleracaoMesaForno: DINT;
	dAccMesaForno: DINT;
	dDecMesaForno: DINT;
	///Contador muda posição de parada do VaiVem
	ContadorMudaPos: INT;
	///Variaveis que Habilitam o Inicio do Ciclo de Aquecimento
	///Variáveis Booleanas Auxiliares
	xFimTempoPausaRoletes: BOOL;
	xFimTempoAquecForno: BOOL;
	xFinalizaVaivemForno: BOOL;
	xFimCalculoCarga: BOOL;
	xTamanhoCargaFora: BOOL;
	xTamanhoCargaOk: BOOL;
	xReativaVaivem: BOOL;
	///Variáveis inteiras Auxiliares
	dValEncoVelMinForno: DINT;
	dValEncoCargaForno: DINT;
	dValEncoAvancoForno: DINT;
	dValEncoRecuoForno: DINT;
	dValEncoDescargaForno: DINT;
	dValEncoReferenciaResfriador: DINT;
	dValEncoSemEnergia: DINT;
	dValLiberaCargaForno: DINT;
	dTamanhoAreaUtilForno: DINT;
	dTamanhoMaximoCarga: DINT;
	dTamanhoCarga: DINT;
	///Distancia Restante para o fim do Carregamento (milimetro)
	iValorVelMinimaForno: INT;
	iValorCargaForno: INT;
	iValorOscilacaoForno: INT;
	iValorDescargaForno: INT;
	iTamanhoAreaUtilForno: INT;
	iValMilimetroVelMinForno: INT;
	iValMilimetroCargaForno: INT;
	iValMilimetroAvancoForno: INT;
	iValMilimetroRecuoForno: INT;
	iValMilimetroDescargaForno: INT;
	iValMilimetroAreaUtilForno: INT;
	iValMilimetroTamMaxCarga: INT;
	iValMilimetroReferenciaResfriador: INT;
	xSensorEntradaPo: BOOL;
	PulsoPoSensorEntrada: PulsoPositivo;
	xliberaDescargaForno: BOOL;
	xDelayMovForno: BOOL;
	xForceSaidadoVidro: BOOL;
	///Variáveis internas auxiliares para mundaça de Velocidade e Posição
	dValorAvancoForno: DINT;
	///////////////
	dValorRecuoForno: DINT;
	////////////////
	xVelocidade01VaivemForno: BOOL;
	//////
	xPosicao01VaivemForno: BOOL;
	/////////
	xFimTempoTrocaVelocidade: BOOL;
	//////
	xFimTempoTrocaPosicao: BOOL;
	//////
	xTemperaturaDesliga: BOOL;
	xDesligaMotorForno: BOOL;
	xTempoMvFornoIn: BOOL;
	xTempoMvFornoQ: BOOL;
	TempoMvForno: ton;
	rConsumoInicialCarga_kW: REAL;
END_VAR

//SELEÇÃO DOS PARAMETROS PELA ESPESSURA DO VIDRO
// Parametros de medidas do Forno
SelecaoPulsos(
	xSelecao:= xEspessuraVidroFino,
	iEntrada0101:= iValorVelMinimaFornoVidroFin,
	iEntrada0102:= iValorVelMinimaFornoVidroGro,
	iEntrada0201:= iValorCargaFornoVidroFin,
	iEntrada0202:= iValorCargaFornoVidroGro,
	iEntrada0301:= iValorOscilacaoFornoVidroFin,
	iEntrada0302:= iValorOscilacaoFornoVidroGro,
	iEntrada0401:= iValorDescargaFornoVidroFin,
	iEntrada0402:= iValorDescargaFornoVidroGro,
	iEntrada0501:= iTamanhoAreaUtilFornoVidroFin,
	iEntrada0502:= iTamanhoAreaUtilFornoVidroGro,
	iEntrada0601:= iTamanhoCargaMaxFornoVidroFin,
	iEntrada0602:= iTamanhoCargaMaxFornoVidroGro,
	iEntrada0701:= iTamanahoFornoContratoVidroFin,
	iEntrada0702:= iTamanahoFornoContratoVidroGro,
	iSaida01=> iValorVelMinimaForno,
	iSaida02=> iValorCargaForno,
	iSaida03=> iValorOscilacaoForno,
	iSaida04=> iValorDescargaForno,
	iSaida05=> iTamanhoAreaUtilForno,
	iSaida06=> iTamanhoCargaMaxForno,
	iSaida07=> iTamanhoCargaContrato);

//Parametros de Rampas do Inversor
//Aceleração
IF 	xEspessuraVidroFino THEN
	dAccMesaForno:=dAccMesaFornoVidroFin;
	dDecMesaForno:=dDecMesaFornoVidroFin;
ELSE
	dAccMesaForno:=dAccMesaFornoVidroGro;
	dDecMesaForno:=dDecMesaFornoVidroGro;
END_IF

IF (dAccMesaForno<>dAceleracaoMesaForno) OR (dDecMesaForno<>dDesaceleracaoMesaForno) THEN
	dAceleracaoMesaForno:=dAccMesaForno;
	dDesaceleracaoMesaForno:=dDecMesaForno;
	xExecutaSetRampasForno:=TRUE;
ELSE
	xExecutaSetRampasForno:=FALSE;
END_IF

// CALCULOS DE POSICIONAMENTO
CalculosMesaForno(
	DistanciaVelMinForno:= 	iValorVelMinimaForno,
	DistanciaCargaForno:= 	iValorCargaForno,
	TamanhoAreaUtil:= 		iTamanhoAreaUtilForno,
	TamanhoCargaMaxima:= 	iTamanhoCargaMaxForno,
	TamanhoCarga:= 			iTamanhoCargaAtualForno,
	SetPointVelMinCarga=> 	iValMilimetroVelMinForno,
	SetPointCargaForno=> 	iValMilimetroCargaForno,
	SetPointDescargaForno=> iValMilimetroDescargaForno,
	SetPointAvancaVaiVemForno=> iValMilimetroAvancoForno,
	SetPointRecuaVaiVemForno=> iValMilimetroRecuoForno,
	TamanhoAreaUtilForno=> 	iValMilimetroAreaUtilForno,
	TamanhoCargaMaxForno=> 	iValMilimetroTamMaxCarga);

// CONVERSÃO MILIMETROS EM PULSOS

iValMilimetroReferenciaResfriador:=iValDistanciaReferenciaResfriador;

ConversorMilimPul(
	dPulso:= 82071,
	dMilimetro:= 6192,
	iEntrMilimetro01:= iValMilimetroVelMinForno,
	iEntrMilimetro02:= iValMilimetroCargaForno,
	iEntrMilimetro03:= iValMilimetroAvancoForno,
	iEntrMilimetro04:= iValMilimetroRecuoForno,
	iEntrMilimetro05:= iValorDescargaForno,//iValMilimetroDescargaForno,
	iEntrMilimetro06:= iValMilimetroAreaUtilForno,
	iEntrMilimetro07:= iValMilimetroTamMaxCarga,
	iEntrMilimetro08:= 40,
	iEntrMilimetro09:= iValMilimetroReferenciaResfriador,
	iEntrMilimetro10:= 400,//distancia da porta de saida para liberar a carga
	dSaidaPulso01=> dValEncoVelMinForno,
	dSaidaPulso02=> dValEncoCargaForno,
	dSaidaPulso03=> dValEncoAvancoForno,
	dSaidaPulso04=> dValEncoRecuoForno,
	dSaidaPulso05=> dValEncoDescargaForno,
	dSaidaPulso06=> dTamanhoAreaUtilForno,
	dSaidaPulso07=> dTamanhoMaximoCarga,
	dSaidaPulso08=>	dValEncoSemEnergia,
	dSaidaPulso09=> dValEncoReferenciaResfriador,
	dSaidaPulso10=> dValLiberaCargaForno);

// CALCULO DO TAMANHO DA CARGA

PulsoPoSensorEntrada(Entrada:= xSensorEntrada, SaidaPulsoPo=>xSensorEntradaPo );

IF	xSensorEntradaPo AND xIniciaCargaMesaEntrada THEN
	xIniciaCargaForno:=TRUE;
	xIniciaCargaMesaEntrada:=FALSE;
END_IF

TamanhoCarga(
	Sensor:= xSensorEntrada,
	Habilita:= xCarregandoForno,
	ValEncoder:= dValorEncoderForno,
	FimMedicao:= xFimCalculoCarga,
	TamanhoCarga=> dTamanhoCarga);

// Desligamento pela Temperatura

IF rMediaLogicaTemperaturaTotal< 0 THEN
	xTemperaturaDesliga:=TRUE;
ELSE
	xTemperaturaDesliga:=FALSE;
END_IF

IF xTemperaturaDesliga AND NOT xResistenciasLigadas THEN
	xDesligaMotorForno:=TRUE;
	xDesligaMotorFornoTempBaixa:=TRUE;
ELSE
	xDesligaMotorForno:=FALSE;
	xDesligaMotorFornoTempBaixa:=FALSE;
END_IF

// MOVIMENTAÇÃO DA MESA DO FORNO
// Atrase para iniciar motor após habilitação
TonDelayMovForno(IN:= xInvMesaFornoHabilitado, PT:=T#1S , Q=> xDelayMovForno, ET=> );
TempoMvForno(IN:= xTempoMvFornoIn, PT:=T#2S , Q=> xTempoMvFornoQ, ET=> );

// Movimentação Stand-By
CASE PassoIniciaForno OF

	0:	(*IF xDelayMovForno THEN
			xLedStart:=TRUE;
		END_IF
		IF xRestart THEN
			PassoIniciaForno:=1;
		END_IF

	1:*)  xLedStart:=FALSE;
		IF NOT xFornoEmCicloComCarga (*AND xDelayMovForno AND NOT xErroEixoMf*) AND NOT xOperacaoManual THEN
			PassoIniciaForno:=2;
			PassoManualForno:=0;
		END_IF

	2:	TonIniVelStdIn:=TRUE;
		IF TonIniVelStdQ THEN
			PassoIniciaForno:=3;
		END_IF

	3:	TonIniVelStdIn:=FALSE;
		PassoIniciaForno:=5;

	5:  iVelocidadeMesaForno:= iVelocidadeStbForno;(*Velocidade Stand-By Forno*)
		PassoIniciaForno:=10;

	10:	xAvancoMesaForno:=TRUE;
		PassoIniciaForno:=15;

	15:	IF iVelocidadeMesaForno<> iVelocidadeStbForno THEN
			PassoIniciaForno:=5;
		END_IF
		IF xFornoEmCicloComCarga THEN
			PassoIniciaForno:=20;
		END_IF
		IF	xDesligaMotorForno THEN
			PassoIniciaForno:=100;
		END_IF
		IF xSemEnergia THEN
			PassoIniciaForno:=50;
		END_IF
		IF xPause THEN
			PassoPauseIniForno:=5;
			PassoIniciaForno:=300;
		END_IF
		IF xAlarmeMotorForno THEN
			PassoAlmIniForno:=5;
			PassoIniciaForno:=400;
		END_IF

	20: IF NOT xFornoEmCicloComCarga THEN
			PassoIniciaForno:=0;
		END_IF

	50: xAvancoMesaForno:=FALSE;
		PassoIniciaForno:=55;

	55: PassoIniciaForno:=60;

	60:	TonParadaSemEnerIn:=TRUE;
		IF TonParadaSemEnerQ THEN
			PassoIniciaForno:=63;
		END_IF
		IF xEnergiaOk THEN
			PassoIniciaForno:=90;
		END_IF

	63:	TonParadaSemEnerIn:=FALSE;
		xHomeEncoderForno:=TRUE;
		PassoIniciaForno:=64;

	64: iVelocidadeMesaForno:= iVelocidadeStbForno;(*Velocidade Stand-By Forno*)
		PassoIniciaForno:=65;

	65:	xHomeEncoderForno:=FALSE;
		PassoIniciaForno:=70;

	70:	xAvancoMesaForno:=TRUE;
		PassoIniciaForno:=75;

	75: IF (dValorEncoderForno>=dValEncoSemEnergia) THEN
			PassoIniciaForno:=50;
		END_IF

	90:	TonParadaSemEnerIn:=FALSE;
		PassoIniciaForno:=0;

	100:xAvancoMesaForno:=FALSE;
		PassoIniciaForno:=105;

	105: PassoIniciaForno:=110;

	110: IF NOT xDesligaMotorForno THEN
		    PassoIniciaForno:=0;
	     END_IF

	// Emergência Pausa/Reinicio
	300:xAvancoMesaForno:=FALSE;
		PassoIniciaForno:=301;

	301:PassoIniciaForno:=302;

	302:IF xRestart THEN
			PassoIniciaForno:=303;
		END_IF

	303:PassoIniciaForno:=PassoPauseIniForno;

		// Alarme Motor Parada/Reinicio

	400:xAvancoMesaForno:=FALSE;
		PassoIniciaForno:=401;

	401:TonAutoResetMotorFornoIn:=TRUE;
		IF TonAutoResetMotorFornoQ THEN
			PassoIniciaForno:=402;
		END_IF

	402: xAutoResetMotorForno:=TRUE;
		PassoIniciaForno:=403;

	403: TonAutoResetMotorFornoIn:=FALSE;
		 PassoIniciaForno:=404;

	404:IF (xRestart OR xAutoResetMotorForno) AND iCanOpenInverMesaFornoStateOk  THEN
			xAutoResetMotorForno:=FALSE;
			PassoIniciaForno:=PassoAlmIniForno;
		END_IF

END_CASE
TonAutoResetMotorForno(IN:=TonAutoResetMotorFornoIn , PT:=T#1000MS , Q=>TonAutoResetMotorFornoQ , ET=> );

TonIniVelStd(IN:=TonIniVelStdIn , PT:=T#100MS , Q=>TonIniVelStdQ , ET=> );
TonParadaSemEner(IN:=TonParadaSemEnerIn , PT:=T#1M , Q=>TonParadaSemEnerQ , ET=>TonParadaSemEnerEt );

iTempoPassoSemEnerg:= DINT_TO_INT((TIME_TO_DINT(T#1M))/1000-(TIME_TO_DINT(TonParadaSemEnerEt))/1000);

// Condição para Descarga do Forno
xliberaDescargaForno:= (xAvancandMesaResfriador AND xFinalizaVaivemForno AND xResfriadorVazio(*AND xDuctosSup01CheckOk AND xGuilhotina01CheckOk AND xVelocidadeVentilador01Ok AND xVelocidadeVentilador02Ok AND xVelocidadeVentilador03Ok*)) OR xForceSaidadoVidro;

// Movimentação em Ciclo
// Sequencia de mudança de Velocidade de VaiVem
CASE PassoVelVaivem OF
	0:	IF xVelocidade01VaivemForno THEN
			PassoVelVaivem:=5;
		END_IF

	5:	xVelocidade01VaivemForno:=FALSE;
		PassoVelVaivem:=10;

	10:	iVelocidadeVaiVemMesaForno := REAL_TO_INT(iVelocidade01Vaivem/10);
		IF xFimTempoTrocaPosicao THEN
			PassoVelVaivem:=15;
		END_IF

	15:	iVelocidadeVaiVemMesaForno:= REAL_TO_INT(iVelocidade02Vaivem/10);
		IF xFimTempoTrocaVelocidade THEN
			PassoVelVaivem:=20;
		END_IF

	20: iVelocidadeVaiVemMesaForno:=REAL_TO_INT(iVelocidade03Vaivem/10);
		//PassoVelVaivem:=20;

	//20:	PassoVelVaivem:=0;
END_CASE

// Sequencia de mudança de Posicao de VaiVem
CASE PassoPosVaivem OF
	0:	IF xPosicao01VaivemForno THEN
			PassoPosVaivem:=5;
		END_IF

	5:	xPosicao01VaivemForno:=FALSE;
		PassoPosVaivem:=10;

	10:	IF NOT xFimTempoTrocaPosicao THEN
			IF ContadorMudaPos=0 THEN
				dValorAvancoForno:= dValEncoCargaForno;
				dValorRecuoForno:= dValEncoCargaForno-773;//Recua 50mm
			END_IF
			IF ContadorMudaPos=1 THEN
				dValorAvancoForno:= dValEncoCargaForno-154;// Avança com -10mm da posição inicial
				dValorRecuoForno:= dValEncoCargaForno-927;//Recua 60mm
			END_IF
			IF ContadorMudaPos=2 THEN
				dValorAvancoForno:= dValEncoCargaForno-309;// Avança com -20mm da posição inicial
				dValorRecuoForno:= dValEncoCargaForno-1081;//Recua 70mm;
			END_IF
			IF ContadorMudaPos=3 THEN
				dValorAvancoForno:= dValEncoCargaForno-463;// Avança com -30mm da posição inicial
				dValorRecuoForno:= dValEncoCargaForno-1235;//Recua 80mm;
			END_IF
		ELSE
			xTempoPausaRoletesOn:=FALSE;
			PassoPosVaivem:=15;
		END_IF

	15:	IF ContadorMudaPos=0 THEN
			dValorAvancoForno:= dValEncoAvancoForno;
			dValorRecuoForno:= dValEncoRecuoForno;
		END_IF
		IF ContadorMudaPos=1 THEN
			dValorAvancoForno:= dValEncoAvancoForno-154;
			dValorRecuoForno:= dValEncoRecuoForno-154;
		END_IF
		IF ContadorMudaPos=2 THEN
			dValorAvancoForno:= dValEncoAvancoForno-309;
			dValorRecuoForno:= dValEncoRecuoForno-309;
		END_IF
		IF ContadorMudaPos=3 THEN
			dValorAvancoForno:= dValEncoAvancoForno-463;
			dValorRecuoForno:= dValEncoRecuoForno-463;
		END_IF
		//PassoPosVaivem:=0;

END_CASE

// Sequencia de Entrada, Oscilação e Saída

CASE PassoMesaForno OF

	0:	IF xIniciaCargaForno AND xFornoEmCiclo THEN
			PassoMesaForno:=1;
		END_IF

	1:	xHomeEncoderForno:=TRUE;
		PassoMesaForno:=2;

	2:	xMesaFornoOn:=TRUE;
		PassoMesaForno:=5;

	5:	xHomeEncoderForno:=FALSE;
		PassoMesaForno:=6;

	6:	iVelocidadeMesaForno:= iVelocidadeCargaMesaForno;(*Velocidade Carga Forno*)
		PassoMesaForno:=7;

	7:	xAvancoMesaForno:=TRUE;
		PassoMesaForno:=10;

	10:	xIniciaCargaForno:=FALSE;
		xIniciaCargaMesaEntrada:=FALSE;
		xExecutaMovMesaForno:=FALSE;
		//xPortaEntradaForno:=TRUE;
		xCarregandoForno:=TRUE;
		xStartCargaForno:=TRUE;
		xFornoCheio:=TRUE;
		PassoMesaForno:=20;

	20: IF (dValorEncoderForno>=dValEncoVelMinForno) THEN
			PassoMesaForno:=30;
		END_IF
		IF xPause THEN
			PassoPauseForno:=5;
			PassoMesaForno:=300;
		END_IF
		IF xAlarmeMotorEntrada OR xAlarmeMotorForno OR xAlarmeGeralEncoderMeForno OR xAlarmePortaEntradaForno THEN
			PassoAlmMesaForno:=5;
			PassoMesaForno:=400;
		END_IF

	30: iVelocidadeMesaForno:= iVelMinCargaForno;(*Velocidade Minima Carga Forno*)
		PassoMesaForno:=40;

	40: IF (dValorEncoderForno>=dValEncoCargaForno) THEN
			PassoMesaForno:=42;
		END_IF
		IF xPause THEN
			PassoPauseForno:=5;
			PassoMesaForno:=300;
		END_IF
		IF xAlarmeMotorForno THEN
			PassoAlmMesaForno:=5;
			PassoMesaForno:=400;
		END_IF

	42: iVelocidadeMesaForno:= 0;
		xAvancoMesaForno:=FALSE;
		PassoMesaForno:=45;

	45: IF (iVelocidade01Vaivem=0) AND (iTempoPosicaoForno<>0)THEN
			xTempoPausaRoletesOn:=TRUE;
		END_IF
		PassoMesaForno:=50;

	50: xExecutaMovMesaForno:=FALSE;
		xCarregandoForno:=FALSE;
		xIniciaCargaForno:=FALSE;
		xFimCarregamentoMesaEntrada:=TRUE; //-> TASK/MesaEntrada
		PassoMesaForno:=55;

	55: IF xFimCalculoCarga THEN
			PassoMesaForno:=60;
		END_IF

	60:	IF (dTamanhoCarga>=dTamanhoAreaUtilForno) OR (dTamanhoCarga>dTamanhoMaximoCarga) OR (dTamanhoCarga<=0) OR  (xSensorEntrada) THEN
			xTamanhoCargaFora:=TRUE;
			xRetornaMesaEntrada:=TRUE; //-> TASK/MesaEntrada
			PassoMesaForno:=70;
		END_IF
		IF (dTamanhoCarga<=dTamanhoMaximoCarga) AND NOT xSensorEntrada THEN
			xTamanhoCargaOk:=TRUE;
			xFimCargaMesaEntrada:=TRUE;//-> TASK/MesaEntrada
			PassoMesaForno:=100;
		END_IF

	70:	xTamanhoCargaFora:=FALSE;
		iVelocidadeMesaForno:= 1*iVelocidadeCargaMesaForno;(*iVelRetornoCargaForno;Velocidade de Retorno Forno*)
		PassoMesaForno:=71;

	71:	xRecuoMesaForno:=TRUE;
		PassoMesaForno:=80;

	80:	xRetornandoForno:=TRUE;
		xExecutaMovMesaForno:=FALSE;
		xTempoPausaRoletesOn:=FALSE;
		IF (dValorEncoderForno<=0) THEN
			PassoMesaForno:=90;
		END_IF
		IF xPause THEN
			PassoPauseForno:=70;
			PassoMesaForno:=300;
		END_IF
		IF xAlarmeMotorEntrada OR xAlarmeMotorForno OR xAlarmeGeralEncoderMeForno OR xAlarmePortaEntradaForno THEN
			PassoAlmMesaForno:=70;
			PassoMesaForno:=400;
		END_IF

	90: xFimRetornoMesaEntrada:=TRUE; //-> TASK/MesaEntrada
		xRecuoMesaForno:=FALSE;		(* DesLiga Recuo Motor Pre Forno *)
		xRetornandoForno:=FALSE;
		xFornoCheio:=FALSE;
		xFornoEmCicloComCarga:=FALSE;
		xPortaEntradaForno:=FALSE;
		xMesaFornoOn:=FALSE;
		PassoIniciaForno:=20;
		PassoMesaForno:=0;

	100: uNumeroCargaRel:=uNumeroCargaRel+1;
		 rConsumoInicialCarga_kW:=rConsumoEnergiaReal_kWh;(*Ativo*)
		 PassoMesaForno:=101;

	101:xIniciaRelatorioProd:=TRUE;
		PassoMesaForno:=102;

	102: xTamanhoCargaOk:=FALSE;
		 xPortaEntradaForno:=FALSE;
		 xFornoCarregado:= TRUE;
		 xFornoComCarga:=TRUE;
		 xIniciaPausaResistencias:= TRUE;
		 xPausaHabilitaTesteEncoder:=TRUE;
		 xLigaConveccaoForno:= TRUE;
		 xVelocidade01VaivemForno:=TRUE;////////
		 xPosicao01VaivemForno:=TRUE;///////////
		 PassoMesaForno:=110;

	110://IF 	xFimTempoPausaRoletes THEN
			PassoMesaForno:=120;
		//END_IF
		IF xPause THEN
			PassoPauseForno:=110;
			PassoMesaForno:=300;
		END_IF
		IF xAlarmeMotorForno THEN
			PassoAlmMesaForno:=110;
			PassoMesaForno:=400;
		END_IF

	120:IF ContadorMudaPos>=4 THEN
			 ContadorMudaPos:=0;
		END_IF
		PassoMesaForno:=121;

	121:xPausaHabilitaTesteEncoder:=FALSE;
		iVelocidadeMesaForno:= 1*iVelocidadeVaiVemMesaForno;(*Velocidade Vai Vem Forno*)
		PassoMesaForno:=122;

	122:xRecuoMesaForno:=TRUE;
		PassoMesaForno:=130;

	130:PassoMesaForno:=135;

	135:IF NOT xliberaDescargaForno OR xAlarmePortaSaidaFornoAberta THEN
			IF (dValorEncoderForno<=dValorRecuoForno) THEN
				PassoMesaForno:=140;
			END_IF
			IF iVelocidadeMesaForno <> 1*iVelocidadeVaiVemMesaForno THEN
				PassoMesaForno:=121;
			END_IF
			IF xPause THEN
				PassoPauseForno:=121;
				PassoMesaForno:=300;
			END_IF
			IF xAlarmeMotorForno OR xAlarmeGeralEncoderMeForno THEN
				PassoAlmMesaForno:=121;
				PassoMesaForno:=400;
			END_IF
		ELSE
			IF	(dValorEncoderForno<=dValEncoCargaForno - dValLiberaCargaForno) THEN
					PassoMesaForno:=156;
			END_IF
			IF iVelocidadeMesaForno <> 1*iVelocidadeVaiVemMesaForno THEN
				PassoMesaForno:=121;
			END_IF
			IF xPause THEN
				PassoPauseForno:=121;
				PassoMesaForno:=300;
			END_IF
			IF xAlarmeMotorForno OR xAlarmeGeralEncoderMeForno THEN
				PassoAlmMesaForno:=121;
				PassoMesaForno:=400;
			END_IF
		END_IF

	140:xRecuoMesaForno:=FALSE;
		PassoMesaForno:=141;

	141:xForceSaidadoVidro:=FALSE;
		PassoMesaForno:=145;

	145:iVelocidadeMesaForno:= iVelocidadeVaiVemMesaForno;(*Velocidade Vai Vem Forno*)
		PassoMesaForno:=146;

	146:xAvancoMesaForno:=TRUE;
		PassoMesaForno:=150;

	150:PassoMesaForno:=151;

	151:IF NOT xliberaDescargaForno OR xAlarmePortaSaidaFornoAberta THEN
			IF (dValorEncoderForno>=dValorAvancoForno) THEN
				PassoMesaForno:=155;
			END_IF
			IF iVelocidadeMesaForno <> 1*iVelocidadeVaiVemMesaForno THEN
				PassoMesaForno:=145;
			END_IF
			IF xPause THEN
				PassoPauseForno:=145;
				PassoMesaForno:=300;
			END_IF
			IF xAlarmeMotorForno OR xAlarmeGeralEncoderMeForno THEN
				PassoAlmMesaForno:=145;
				PassoMesaForno:=400;
			END_IF
		ELSE
			IF	(dValorEncoderForno<=dValEncoCargaForno - dValLiberaCargaForno) THEN
				PassoMesaForno:=157;
			ELSE
				PassoMesaForno:=155;
			END_IF
			IF iVelocidadeMesaForno <> 1*iVelocidadeVaiVemMesaForno THEN
				PassoMesaForno:=145;
			END_IF
			IF xPause THEN
				PassoPauseForno:=145;
				PassoMesaForno:=300;
			END_IF
			IF xAlarmeMotorForno OR xAlarmeGeralEncoderMeForno THEN
				PassoAlmMesaForno:=145;
				PassoMesaForno:=400;
			END_IF
		END_IF

	155: xAvancoMesaForno:=FALSE;
		 ContadorMudaPos:=ContadorMudaPos+1;
		 PassoMesaForno:=120;

	156:xRecuoMesaForno:=FALSE;
		xAvancoMesaForno:=TRUE;
		xForceSaidadoVidro:=FALSE;
		PassoMesaForno:=157;

	157:xForceSaidadoVidro:=FALSE;
		PassoMesaForno:=160;

	160://xForceSaidadoVidro:=FALSE;
		PassoMesaForno:=164;

	164:xAvancoMesaForno:=TRUE;
		PassoMesaForno:=165;

	165:iVelocidadeMesaForno:= iVelocidadeDescargaMesaForno;(*Velocidade Descarga Forno*)
		PassoMesaForno:=166;

	166:PassoMesaForno:=170;

	170:IF xDescarregandoForno THEN
			PassoMesaForno:=180;
		ELSE
			PassoMesaForno:=171;
		END_IF

	171:xAbreVenezVentPass:=TRUE;//-> TASK/T_VenezianaVentInfPass
		xPortaSaidaForno:=TRUE;
		xValvulaScanner:=TRUE;
		xDescarregandoForno:=TRUE;
		//xReajustaAlturaDuctosSup02:=TRUE;
		xFornoCarregado:= FALSE;
		xPulsoTrocaParamResfriador:=TRUE;
		xIniciaPausaResistencias:= FALSE;
		xLigaConveccaoForno:= FALSE;
		PassoMesaForno:=172;

	172:IF (dValorEncoderForno>=dValEncoCargaForno) AND xSensorPortaSaida THEN
			PassoMesaForno:=175;
		END_IF
		IF (dValorEncoderForno>=dValEncoCargaForno) AND NOT xSensorPortaSaida THEN
			PassoMesaForno:=173;
		END_IF
		IF xPause THEN
			xDescarregandoForno:=FALSE;
			xFornoCarregado:= TRUE;
			PassoPauseForno:=121;
			PassoMesaForno:=300;
		END_IF
		(*IF xAlarmeMeFornoParado THEN // Só funciona se resetar Este alarme
			xDescarregandoForno:=FALSE;
			xFornoCarregado:= TRUE;
			PassoMesaForno:=121;
		END_IF*)

	173: xDescarregandoForno:=FALSE;
		 xFornoCarregado:= TRUE;
		 xAvancoMesaForno:=FALSE;
		 PassoMesaForno:=120;

	175: //xValvulaScanner:=TRUE;
		 PassoMesaForno:=176;

	176: xFimTempoPausaRoletes:=FALSE;
		 xFimTempoAquecForno:=FALSE;
		 xFinalizaVaivemForno:=FALSE;
		 xFimTempoTrocaVelocidade:=FALSE;//////
		 xFimTempoTrocaPosicao:=FALSE;//////
		 xFimTempoPausaResistInf:=FALSE;
		 xFimTempoPausaResistSup:=FALSE;
		 xFimTempoPausa02ResistSup:=FALSE;
		 PassoVelVaivem:=0;////////
		 PassoPosVaivem:=0;////////
		 PassoMesaForno:=180;

	180:IF (dValorEncoderForno>=dValEncoReferenciaResfriador) THEN
			xIniciaCargaResfriador:=TRUE;//-> TASK/MesaEntrada
			xIniciaCargaPassagem:=TRUE;//-> TASK/MesaEntrada
			PassoMesaForno:=181;
		END_IF
		IF xPause THEN
			PassoPauseForno:=164;
			PassoMesaForno:=300;
		END_IF
		IF xAlarmeMotorForno OR xAlarmeMotorResfriador OR xAlarmePortaSaidaFornoAberta OR xAlarmeGeralEncoderMeForno OR xAlarmeGeralEncoderMeResfriador THEN
			PassoAlmMesaForno:=164;
			PassoMesaForno:=400;
		END_IF

	181:IF (dValorEncoderForno>=dValEncoDescargaForno) THEN
			PassoMesaForno:=190;
		END_IF
		IF xPause THEN
			PassoPauseForno:=164;
			PassoMesaForno:=300;
		END_IF
		IF xAlarmeMotorForno OR xAlarmeMotorResfriador OR xAlarmePortaSaidaFornoAberta OR xAlarmeGeralEncoderMeResfriador THEN
			PassoAlmMesaForno:=164;
			PassoMesaForno:=400;
		END_IF

	190:xFinalizaRelatorioProd:=TRUE;
		xDescarregandoForno:=FALSE;
		xFornoCheio:=FALSE;
		xFornoComCarga:=FALSE;
		xPortaSaidaForno:=FALSE;
		xValvulaScanner:=FALSE;
		xForceSaidadoVidro:=FALSE;
		xFimDescForIniStdBy:=TRUE;
		xResetPid:=TRUE;
		PassoMesaForno:=191;

	191:IF xCarregamentoHabilitado THEN
			xRecargaForno:=TRUE; //->TASK/MesaEntrada
			xDelayCargaForno:=TRUE; //->TASK/MesaEntrada
			PassoMesaForno:=0;
		ELSE
			xFornoEmCicloComCarga:=FALSE;
			xDelayCargaForno:=TRUE; //->TASK/MesaEntrada
			xMesaFornoOn:=FALSE;
			PassoMesaForno:=0;
		END_IF

	// Emergência Pausa/Reinicio
	300:xAvancoMesaForno:=FALSE;
		xRecuoMesaForno:=FALSE;
		PassoMesaForno:=301;

	301:PassoMesaForno:=302;

	302:IF xRestart THEN
			PassoMesaForno:=303;
		END_IF

	303:PassoMesaForno:=PassoPauseForno;

		// Alarme Motor Parada/Reinicio
	400:xAvancoMesaForno:=FALSE;
		xRecuoMesaForno:=FALSE;
		PassoMesaForno:=401;

	401:PassoMesaForno:=402;

	402:IF (xRestart) AND iCanOpenInverMesaFornoStateOk  THEN
			PassoMesaForno:=PassoAlmMesaForno;
		END_IF

END_CASE

//Consumo de Energia por fornada
rConsumoCargaRel:= rConsumoEnergiaReal_kWh-rConsumoInicialCarga_kW;

TpSairForno(IN:=xBtSairForno , PT:=T#500MS , Q=>xSairForno , ET=> );
IF xBtSairForno THEN
	xBtSairForno:=0;
END_IF

IF xSairForno AND NOT xResfriadorCheio AND xFornoComCarga THEN
	xForceSaidadoVidro:=TRUE;
END_IF

// TEMPORIZADORES
TempoPausaRoletes(
	IniciaTempo:= 	xFornoCarregado,
	AbortaTempo:= 	xSairForno OR xOperacaoManual,
	SetPointTempo:= iTempoPausaRoletes,
	FimTempo:= 		xFimTempoPausaRoletes,
	TempoDecorrido=>iTempoPausaRoleteDecorrido,
	TempoRestante=> iTempoPausaRoleteRestante);

TempoAquecimForno(
	IniciaTempo:= xFornoCarregado,
	AbortaTempo:= xSairForno OR xOperacaoManual,
	SetPointTempo:= iTempoAquecimForno,
	FimTempo:= 		xFimTempoAquecForno,
	TempoDecorrido=>iTempoAquecFornoDecorrido,
	TempoRestante=> iTempoAquecFornoRestante);

xFinalizaVaivemForno:=xFimTempoAquecForno;
xLigaCargaResfriador:=xFimTempoAquecForno;
xLigaCargaPassagem:=xFimTempoAquecForno;
xLigaVent01FimForno:=	xFimTempoAquecForno AND NOT xMotorVentilador01Ligado;
xLigaVent02FimForno:=	xFimTempoAquecForno AND NOT xMotorVentilador02Ligado;
xLigaVent03FimForno:=	xFimTempoAquecForno AND NOT xMotorVentilador03Ligado;
xLigaVent04FimForno:=	xFimTempoAquecForno AND NOT xMotorVentilador04Ligado;

/////////////////////////////////////////////////////
TempoTrocaVelocidade(
	IniciaTempo:= xFimTempoTrocaPosicao,(*xFornoCarregado,*)
	AbortaTempo:= xSairForno OR xOperacaoManual,
	SetPointTempo:= iTempoVelocidadeForno,
	FimTempo:= xFimTempoTrocaVelocidade,
	TempoDecorrido=> iTempoTrocaVelocidadeDecorrido,
	TempoRestante=> );

TempoTrocaPosicao(
	IniciaTempo:= xFornoCarregado,
	AbortaTempo:= xSairForno OR xOperacaoManual,
	SetPointTempo:= iTempoPosicaoForno,
	FimTempo:= xFimTempoTrocaPosicao,
	TempoDecorrido=> iTempoTrocaPosicaoDecorrido,
	TempoRestante=> );

//STATUS
xFornoVazio:=NOT xFornoCheio;

// MOVIMENTAÇÃO PELO COMANDO ENTRADAS DIGITAIS DO INVERSOR
// Comando e Direção
xMotorMesaFornoAvanco:= xAvancoMesaForno;
xMotorMesaFornoRecuo:= xRecuoMesaForno;

InversorMesaForno.i_xAvanco:=xMotorMesaFornoAvanco;
InversorMesaForno.i_xRecuo:=xMotorMesaFornoRecuo;

// Velocidade
InversorMesaForno.i_iFreqRef:=iVelocidadeMesaForno;

//------------------------------------------------------------------------\\

IF	uHoraRealTime=21 AND uMinutoRealTime=0 AND uSegundoRealTime=0 THEN
	uNumeroCargaRel:=0;
END_IF

ConversorPulMilim(
	dPulso:= 82071,
	dMilimetro:= 6192,
	dEntradaPulso01:= dTamanhoCarga,
	iSaidaMilimetro01=> iTamanhoCargaAtualForno );

IF xOperacaoManual THEN
	xLedStart:=FALSE;
	PassoIniciaForno:=0;
	PassoPauseIniForno:=0;
	PassoAlmIniForno:=0;
	PassoMesaForno:=0;
	PassoPauseForno:=0;
	PassoAlmMesaForno:=0;

	PassoVelVaivem:=0;////////
	PassoPosVaivem:=0;///////
	ContadorMudaPos:=0;
	xIniciaCargaForno:=FALSE;
	xHomeEncoderForno:=FALSE;
	xCarregandoForno:=FALSE;
	xFornoCheio:=FALSE;
	xFornoEmCicloComCarga:=FALSE;
	xMesaFornoOn:=FALSE;
	xTamanhoCargaFora:=FALSE;
	xTamanhoCargaOk:=FALSE;
	xRetornandoForno:=FALSE;
	xFornoCarregado:= FALSE;
	xIniciaPausaResistencias:= FALSE;
	xLigaConveccaoForno:= FALSE;
	xFimTempoPausaRoletes:=FALSE;
	xFimTempoAquecForno:=FALSE;
	xFimTempoTrocaVelocidade:=FALSE;//////
	xFimTempoTrocaPosicao:=FALSE;//////
	xFinalizaVaivemForno:=FALSE;
	xFimTempoPausaResistInf:=FALSE;
	xFimTempoPausaResistSup:=FALSE;
	xFimTempoPausa02ResistSup:=FALSE;
	xDescarregandoForno:=FALSE;
	xIniciaRelatorioProd:= FALSE;
	xFinalizaRelatorioProd:= FALSE;
	TonParadaSemEnerIn:=FALSE;
	xTempoPausaRoletesOn:=FALSE;
	xFimCalculoCarga:=FALSE;
	xFornoComCarga:=FALSE;
	xPausaHabilitaTesteEncoder:=FALSE;
	xForceSaidadoVidro:=FALSE;
	xVelocidade01VaivemForno:=FALSE;//////
	xPosicao01VaivemForno:=FALSE;/////////
	xAbreVenezVentPass:=FALSE;
	xValvulaScanner:=FALSE;

	xPortaEntradaForno:=FALSE;
	xPortaSaidaForno:=FALSE;

	xAvancoMesaForno:=FALSE;
	xRecuoMesaForno:=FALSE;
END_IF

xDesabFalhInvMesaForno:= NOT xFornoEmCicloComCarga;

(* ---- G_BufferResfriamento.prg.st ---- *)
PROGRAM G_BufferResfriamento
VAR
	Index: INT;
	iEscreverReceitaResfriamento: INT;
END_VAR

//BUFFER PARAMETROS DO RESFRIAMENTO

(*---------------- SISTEMA NOVO --------------------*)

IF ((sFornoNomedaReceita<>sResfriamentoNomedaReceita) OR xResfriamentoReenvioRec) AND NOT xResfriadorEmCiclo THEN
	iEscreverReceitaResfriamento:=1;
END_IF

IF iEscreverReceitaResfriamento=1 THEN
	xResfriamentoReenvioRec:=0;
	iResfriamentoEspessuraVidro:=iFornoEspessuraVidro;

	// Parametros da Mesa do Resfriador
	rEmissividade:=rBuffer02Emissividade;

	iTempoResfriamento:=iBuffer02TempoResfriamento;
	iTempoTrocaEstagioResfriamento:=iBuffer02TempoTrocaEstagioResfriamento;
	iTempoTrocaEstagio02Resfriamento:=iBuffer02TempoTrocaEstagio02Resfriamento;

	//iVelocidade01Ventilador01:=iBuffer02Velocidade01Ventilador01;
	//iVelocidade02Ventilador01:=iBuffer02Velocidade02Ventilador01;
	//iVelocidade03Ventilador01:=iBuffer02Velocidade03Ventilador01;

	//iVelocidade01Ventilador02:=iBuffer02Velocidade01Ventilador02;
	//iVelocidade02Ventilador02:=iBuffer02Velocidade02Ventilador02;
	//iVelocidade03Ventilador02:=iBuffer02Velocidade03Ventilador02;

	iVelocidade01Ventilador03:=iBuffer02Velocidade01Ventilador03;
	iVelocidade02Ventilador03:=iBuffer02Velocidade02Ventilador03;
	iVelocidade03Ventilador03:=iBuffer02Velocidade03Ventilador03;

	//iVelocidade01Ventilador04:=iBuffer02Velocidade01Ventilador04;
	//iVelocidade02Ventilador04:=iBuffer02Velocidade02Ventilador04;
	//iVelocidade03Ventilador04:=iBuffer02Velocidade03Ventilador04;

	// Parametros Resfriador 01 Inferior
	iValAltura01ResfriadorInf01:=iBuffer02ValAltura01ResfriadorInf01;
	iValAltura02ResfriadorInf01:=iBuffer02ValAltura02ResfriadorInf01;
	iValAltura03ResfriadorInf01:=iBuffer02ValAltura03ResfriadorInf01;

	// Parametros Resfriador 01 Superior
	iValAltura01ResfriadorSup01:=iBuffer02ValAltura01ResfriadorSup01;
	iValAltura02ResfriadorSup01:=iBuffer02ValAltura02ResfriadorSup01;
	iValAltura03ResfriadorSup01:=iBuffer02ValAltura03ResfriadorSup01;
	iVeneziana:=iBuffer02Veneziana;
	iPassagem:=iBuffer02Passagem;

	// Parametros Resfriador 02 Inferior
	iValAltura01ResfriadorInf02:=iBuffer02ValAltura01ResfriadorInf02;
	iValAltura02ResfriadorInf02:=iBuffer02ValAltura02ResfriadorInf02;
	iValAltura03ResfriadorInf02:=iBuffer02ValAltura03ResfriadorInf02;

	// Parametros Resfriador 02 Superior
	iValAltura01ResfriadorSup02:=iBuffer02ValAltura01ResfriadorSup02;
	iValAltura02ResfriadorSup02:=iBuffer02ValAltura02ResfriadorSup02;
	iValAltura03ResfriadorSup02:=iBuffer02ValAltura03ResfriadorSup02;

	// Parametros Guilhotina 01
	iAlturaGhilhotina01:=iBuffer02AlturaGhilhotina01;

	iAlturaGhilhotina01Sup:=iBuffer02AlturaGhilhotina01Sup;
	iAlturaGhilhotina01Inf:=iBuffer02AlturaGhilhotina01Inf;

	// Parametros Guilhotina 02
	iAlturaGhilhotina02:=iBuffer02AlturaGhilhotina02;

	iCorretorCargaMesaResfriador:=iBuffer02CorretorCargaMesaResfriador;
	iVelocidadeVaiVemResfriador:=iBuffer02VelocidadeVaiVemResfriador;
	iVelocidadeDescargaMesadoResfriador:=iBuffer02VelocidadeDescargaMesadoResfriador;
	iCorretorCargaMesaSaida:=iBuffer02CorretorCargaMesaSaida;

	sResfriamentoNomedaReceita:=sFornoNomedaReceita;
	xBtRecAjustaAlturaDuctosSup01:=TRUE;
	xBtRecAjustaAlturaDuctosInf01:=TRUE;
	xBtRecAjustaAlturaDuctosSup02:=TRUE;
	xBtRecAjustaAlturaDuctosInf02:=TRUE;
	xBtRecAjustaGuilhotina01:=TRUE;
	xBtRecAjustaGuilhotina01Sup:=TRUE;
	xBtRecAjustaGuilhotina01Inf:=TRUE;
	xBtRecAjustaGuilhotina02:=TRUE;
	iEscreverReceitaResfriamento:=0;

	IF iVeneziana=1 THEN
		xValvulaVeneziana:=TRUE;
	ELSE
		xValvulaVeneziana:=FALSE;
	END_IF

END_IF

IF iResfriamentoEspessuraVidro = 4 THEN
	xEspessuraVidroFinoResfriador:=TRUE;
ELSE
	xEspessuraVidroFinoResfriador:=FALSE;
END_IF

(* ---- G_BufferTemperaPass.prg.st ---- *)
PROGRAM G_BufferTemperaPass
VAR
	iEscreverReceitaPassagem: INT;
END_VAR

IF ((sFornoNomedaReceita<>sResfriamentoNomedaReceita) OR xPassagemReenvioRec) AND NOT xPassandoTempera THEN
	iEscreverReceitaPassagem:=1;
END_IF

IF iEscreverReceitaPassagem=1 THEN
	xPassagemReenvioRec:=0;

	//iVelocidade01Ventilador01:=iBuffer02Velocidade01Ventilador01;
	//iVelocidade02Ventilador01:=iBuffer02Velocidade02Ventilador01;
	//iVelocidade03Ventilador01:=iBuffer02Velocidade03Ventilador01;

	iVelocidade01Ventilador02:=iBuffer02Velocidade01Ventilador02;
	iVelocidade02Ventilador02:=iBuffer02Velocidade02Ventilador02;
	iVelocidade03Ventilador02:=iBuffer02Velocidade03Ventilador02;

	iEscreverReceitaPassagem:=0;
END_IF

(* ---- H1_Dutos_Oscilantes.prg.st ---- *)
PROGRAM H1_Dutos_Oscilantes
VAR
	AlarmeMotorOscilaSup02	: AlarmeMotor ;
	AlarmeMotorOscilaInf02	: AlarmeMotor ;

	TofChAbreDuctosResfrSup02 : TOF ;
	xDlyChAbreDuctosResfrSup02	: bool ;

END_VAR

TofChAbreDuctosResfrSup02(IN:=xChAbreDuctosResfriadorSup02 , PT:=T#3S , Q=>xDlyChAbreDuctosResfrSup02 , ET=> );

xMotorOscilaResfr02Sup:=(xMesaResfriadorOn OR xForceDut) AND NOT xMotorDifusorSup02Ligado AND NOT xDlyChAbreDuctosResfrSup02;
xMotorOscilaResfr02Inf:=(xMesaResfriadorOn OR xForceDut) AND NOT xMotorDifusorSup02Ligado AND NOT xDlyChAbreDuctosResfrSup02;

AlarmeMotorOscilaSup02(
	KaMotor:= xKaMotorOscilaResfr02Sup,
	KmMotor:= xMotorOscilaResfr02Sup,
	ResetAlarm:= bResetAlmGeral,
	AlarmeMotor=> xAlarmeMotorOscilaSup02,
	AlarmeSonoro=> );

AlarmeMotorOscilaInf02(
	KaMotor:= xKaMotorOscilaResfr02Inf,
	KmMotor:= xMotorOscilaResfr02Inf,
	ResetAlarm:= bResetAlmGeral,
	AlarmeMotor=> xAlarmeMotorOscilaInf02,
	AlarmeSonoro=> );

(* ---- H_MesaPassagem.prg.st ---- *)
PROGRAM H_MesaPassagem
VAR
///Passo da Execução da Movimentação do Mesa Passagem
	PassoMesaPassagem: INT;
	PassoPausePassagem: INT;
	PassoAlmMesaPassagem: INT;

	iVelocidadeMesaPassagem: INT;
END_VAR

// MOVIMENTAÇÃO DA MESA DE PASSAGEM

CASE PassoMesaPassagem OF

		0:	IF xLigaCargaPassagem THEN
				PassoMesaPassagem:=1;
			END_IF

		1:	xMesaPassagemOn:=TRUE;
			IF xPause THEN
				PassoPausePassagem:=1;
				PassoMesaPassagem:=300;
				xLigaCargaPassagem:=TRUE;
			ELSIF xAlarmeMotorResfriador THEN
				PassoAlmMesaPassagem:=1;
				PassoMesaPassagem:=400;
			ELSE
				PassoMesaPassagem:=3;
			END_IF

		3:	iVelocidadeMesaPassagem:= iVelocidadeCargaMesaPass;(*Velocidade Carga Resfriador*)
			PassoMesaPassagem:=5;

		5:	xAvancoMesaPassagem:=TRUE;
			PassoMesaPassagem:=8;

		8:	xLigaCargaPassagem:=FALSE;
			IF xIniciaCargaPassagem THEN
				PassoMesaPassagem:=10;
			END_IF
			IF xPause THEN
				PassoPausePassagem:=1;
				PassoMesaPassagem:=300;
				xLigaCargaPassagem:=TRUE;
			END_IF
			IF xAlarmeMotorResfriador THEN
				PassoAlmMesaPassagem:=1;
				PassoMesaPassagem:=400;
			END_IF

		10:  xIniciaCargaPassagem:=FALSE;
			PassoMesaPassagem:=12;

		12:	IF xFimDescargaMesaPass THEN
				PassoMesaPassagem:=14;
		    END_IF

		14: xFimDescargaMesaPass:=FALSE;
			xAvancoMesaPassagem:=FALSE;
			xMesaPassagemOn:=FALSE;
			PassoMesaPassagem:=0;

END_CASE

// MOVIMENTAÇÃO PELO COMANDO ENTRADAS DIGITAIS DO INVERSOR
// Comando e Direção
xMotorMesaPassAvanco:= xAvancoMesaPassagem ;
xMotorMesaPassRecuo:= xRecuoMesaPassagem ;

InversorMesaPass.i_xAvanco:=xMotorMesaPassAvanco;
InversorMesaPass.i_xRecuo:=xMotorMesaPassRecuo;

// Velocidade
InversorMesaPass.i_iFreqRef:=iVelocidadeMesaPassagem;

IF xOperacaoManual THEN
	PassoMesaPassagem:=0;
	PassoPausePassagem:=0;
	PassoAlmMesaPassagem:=0;
	xLigaCargaPassagem:=FALSE;
	xMesaPassagemOn:=FALSE;
	xAvancoMesaPassagem:=FALSE;
	xRecuoMesaPassagem:=FALSE;
END_IF
